C01826=1232.240,4.980,-41.243,-179.381,5.306,148.733
C01827=1232.235,5.230,-41.257,-179.378,5.306,148.732
C01828=1232.230,5.479,-41.273,-179.376,5.307,148.732
C01829=1232.225,5.729,-41.287,-179.373,5.306,148.731
C01830=1232.220,5.979,-41.301,-179.371,5.307,148.730
C01831=1232.215,6.228,-41.316,-179.368,5.308,148.730
C01832=1232.210,6.478,-41.331,-179.366,5.307,148.729
C01833=1232.205,6.727,-41.346,-179.363,5.308,148.728
C01834=1232.200,6.977,-41.361,-179.361,5.308,148.728
C01835=1232.195,7.226,-41.376,-179.358,5.309,148.727
C01836=1232.190,7.476,-41.390,-179.356,5.309,148.726
C01837=1232.185,7.725,-41.405,-179.353,5.309,148.726
C01838=1232.180,7.975,-41.420,-179.351,5.310,148.725
C01839=1232.175,8.224,-41.435,-179.348,5.310,148.724
C01840=1232.170,8.474,-41.450,-179.345,5.310,148.723
C01841=1232.165,8.723,-41.465,-179.343,5.310,148.723
C01842=1232.159,8.973,-41.479,-179.340,5.311,148.722
C01843=1232.155,9.222,-41.494,-179.338,5.311,148.721
C01844=1232.150,9.472,-41.509,-179.335,5.311,148.721
C01845=1232.144,9.721,-41.524,-179.333,5.311,148.720
C01846=1232.140,9.970,-41.539,-179.330,5.312,148.719
C01847=1232.135,10.220,-41.554,-179.328,5.312,148.719
C01848=1232.129,10.469,-41.569,-179.325,5.312,148.718
C01849=1232.124,10.719,-41.583,-179.323,5.313,148.717
C01850=1232.120,10.968,-41.598,-179.320,5.313,148.716
C01851=1232.114,11.217,-41.614,-179.318,5.313,148.716
C01852=1232.109,11.467,-41.628,-179.315,5.314,148.715
C01853=1232.105,11.717,-41.644,-179.313,5.314,148.714
C01854=1232.100,11.967,-41.658,-179.310,5.315,148.714
C01855=1232.095,12.216,-41.673,-179.308,5.314,148.713
C01856=1232.090,12.465,-41.689,-179.305,5.315,148.712
C01857=1232.085,12.715,-41.703,-179.303,5.315,148.712
C01858=1232.079,12.965,-41.719,-179.300,5.316,148.711
C01859=1232.075,13.214,-41.734,-179.298,5.316,148.710
C01860=1232.070,13.463,-41.748,-179.295,5.316,148.710
C01861=1232.064,13.713,-41.764,-179.293,5.317,148.709
C01862=1232.060,13.962,-41.779,-179.290,5.317,148.708
C01863=1232.054,14.212,-41.794,-179.287,5.318,148.708
C01864=1232.050,14.462,-41.809,-179.285,5.318,148.707
C01865=1232.045,14.711,-41.825,-179.283,5.318,148.706
C01866=1232.040,14.960,-41.840,-179.280,5.319,148.705
C01867=1232.034,15.210,-41.854,-179.277,5.319,148.705
C01868=1232.030,15.459,-41.869,-179.275,5.319,148.704
C01869=1232.024,15.709,-41.885,-179.273,5.320,148.703
C01870=1232.020,15.958,-41.900,-179.270,5.320,148.703
C01871=1232.014,16.209,-41.915,-179.267,5.321,148.702
C01872=1232.010,16.458,-41.930,-179.265,5.320,148.701
C01873=1232.004,16.707,-41.946,-179.263,5.321,148.701
C01874=1232.000,16.956,-41.961,-179.260,5.321,148.700
C01875=1231.994,17.206,-41.976,-179.257,5.322,148.699
C01876=1231.989,17.455,-41.991,-179.255,5.322,148.699
C01877=1231.984,17.705,-42.006,-179.253,5.322,148.698
C01878=1231.980,17.954,-42.022,-179.250,5.323,148.697
C01879=1231.975,18.204,-42.037,-179.248,5.324,148.697
C01880=1231.970,18.453,-42.052,-179.245,5.324,148.696
C01881=1231.964,18.703,-42.067,-179.243,5.324,148.695
C01882=1231.960,18.952,-42.082,-179.240,5.324,148.695
C01883=1231.955,19.202,-42.098,-179.238,5.325,148.694
C01884=1231.950,19.451,-42.113,-179.235,5.326,148.693
C01885=1231.945,19.701,-42.129,-179.233,5.325,148.693
C01886=1231.940,19.950,-42.144,-179.230,5.326,148.692
C01887=1231.935,20.199,-42.159,-179.228,5.326,148.691
C01888=1231.930,20.449,-42.175,-179.225,5.327,148.691
C01889=1231.925,20.699,-42.189,-179.223,5.328,148.690
C01890=1231.920,20.948,-42.205,-179.220,5.327,148.689
C01891=1231.915,21.197,-42.220,-179.218,5.328,148.689
C01892=1231.910,21.447,-42.236,-179.215,5.328,148.688
C01893=1231.905,21.697,-42.252,-179.213,5.329,148.687
C01894=1231.900,21.946,-42.267,-179.210,5.329,148.687
C01895=1231.895,22.195,-42.282,-179.208,5.329,148.686
C01896=1231.890,22.445,-42.297,-179.205,5.330,148.685
C01897=1231.885,22.695,-42.313,-179.202,5.330,148.685
C01898=1231.880,22.944,-42.329,-179.200,5.331,148.684
C01899=1231.875,23.193,-42.344,-179.198,5.331,148.683
C01900=1231.870,23.443,-42.359,-179.195,5.331,148.683
C01901=1231.865,23.693,-42.375,-179.192,5.332,148.682
C01902=1231.861,23.942,-42.390,-179.190,5.332,148.681
C01903=1231.855,24.191,-42.406,-179.187,5.333,148.680
C01904=1231.850,24.441,-42.421,-179.185,5.332,148.680
C01905=1231.846,24.690,-42.437,-179.182,5.333,148.679
C01906=1231.840,24.940,-42.452,-179.180,5.334,148.678
C01907=1231.835,25.189,-42.468,-179.177,5.334,148.678
C01908=1231.830,25.438,-42.483,-179.175,5.335,148.677
C01909=1231.825,25.688,-42.499,-179.172,5.334,148.676
C01910=1231.820,25.938,-42.514,-179.170,5.335,148.676
C01911=1231.815,26.187,-42.529,-179.167,5.336,148.675
C01912=1231.811,26.437,-42.545,-179.165,5.336,148.674
C01913=1231.806,26.686,-42.562,-179.162,5.337,148.674
C01914=1231.800,26.935,-42.577,-179.160,5.336,148.673
C01915=1231.796,27.184,-42.592,-179.157,5.337,148.672
C01916=1231.791,27.434,-42.608,-179.155,5.337,148.672
C01917=1231.785,27.684,-42.624,-179.152,5.338,148.671
C01918=1231.780,27.933,-42.639,-179.149,5.339,148.670
C01919=1231.776,28.183,-42.655,-179.147,5.338,148.670
C01920=1231.771,28.432,-42.670,-179.145,5.339,148.669
C01921=1231.765,28.681,-42.687,-179.142,5.339,148.668
C01922=1231.761,28.931,-42.703,-179.140,5.340,148.668
C01923=1231.756,29.180,-42.718,-179.137,5.341,148.667
C01924=1231.750,29.449,-42.735,-179.134,5.341,148.666
C01925=1231.745,29.717,-42.752,-179.131,5.342,148.666
C01926=1231.740,29.986,-42.769,-179.129,5.342,148.665
C01927=1231.734,30.255,-42.786,-179.126,5.343,148.664
C01928=1231.729,30.504,-42.802,-179.124,5.342,148.663
C01929=1231.724,30.753,-42.817,-179.121,5.343,148.663
C01930=1231.720,31.003,-42.833,-179.119,5.344,148.662
C01931=1231.715,31.252,-42.849,-179.116,5.344,148.661
C01932=1231.710,31.502,-42.865,-179.113,5.345,148.661
C01933=1231.704,31.752,-42.880,-179.111,5.345,148.660
C01934=1231.699,32.001,-42.896,-179.109,5.345,148.659
C01935=1231.695,32.250,-42.912,-179.106,5.346,148.659
C01936=1231.690,32.500,-42.928,-179.103,5.346,148.658
C01937=1231.684,32.749,-42.943,-179.101,5.347,148.657
C01938=1231.680,32.999,-42.959,-179.098,5.347,148.657
C01939=1231.675,33.248,-42.976,-179.095,5.348,148.656
C01940=1231.670,33.498,-42.991,-179.093,5.348,148.655
C01941=1231.664,33.748,-43.007,-179.091,5.348,148.655
C01942=1231.660,33.996,-43.023,-179.089,5.349,148.654
C01943=1231.655,34.246,-43.039,-179.086,5.350,148.654
C01944=1231.650,34.496,-43.054,-179.083,5.350,148.653
C01945=1231.645,34.745,-43.071,-179.081,5.351,148.652
C01946=1231.640,34.994,-43.087,-179.079,5.350,148.652
C01947=1231.636,35.244,-43.103,-179.076,5.351,148.651
C01948=1231.630,35.493,-43.119,-179.073,5.352,148.650
C01949=1231.625,35.743,-43.134,-179.071,5.352,148.649
C01950=1231.620,35.992,-43.151,-179.068,5.353,148.649
C01951=1231.615,36.242,-43.167,-179.065,5.353,148.648
C01952=1231.610,36.491,-43.183,-179.063,5.353,148.647
C01953=1231.605,36.740,-43.199,-179.061,5.354,148.647
C01954=1231.600,36.991,-43.215,-179.058,5.354,148.646
C01955=1231.596,37.239,-43.231,-179.055,5.355,148.645
C01956=1231.591,37.488,-43.246,-179.053,5.355,148.645
C01957=1231.586,37.738,-43.263,-179.050,5.356,148.644
C01958=1231.581,37.987,-43.278,-179.047,5.356,148.643
C01959=1231.576,38.237,-43.295,-179.045,5.356,148.643
C01960=1231.571,38.486,-43.311,-179.043,5.357,148.642
C01961=1231.566,38.736,-43.327,-179.041,5.358,148.642
C01962=1231.561,38.985,-43.343,-179.038,5.358,148.641
C01963=1231.556,39.235,-43.360,-179.035,5.359,148.640
C01964=1231.551,39.484,-43.375,-179.033,5.359,148.640
C01965=1231.547,39.733,-43.392,-179.030,5.360,148.639
C01966=1231.541,39.983,-43.407,-179.028,5.360,148.638
C01967=1231.537,40.232,-43.424,-179.025,5.360,148.638
C01968=1231.531,40.482,-43.440,-179.023,5.361,148.637
C01969=1231.526,40.732,-43.457,-179.020,5.361,148.636
C01970=1231.521,40.981,-43.473,-179.017,5.362,148.636
C01971=1231.516,41.230,-43.489,-179.015,5.362,148.635
C01972=1231.511,41.480,-43.505,-179.012,5.363,148.634
C01973=1231.506,41.729,-43.522,-179.010,5.363,148.633
C01974=1231.501,41.978,-43.538,-179.008,5.364,148.633
C01975=1231.496,42.228,-43.554,-179.005,5.364,148.632
C01976=1231.491,42.477,-43.570,-179.003,5.365,148.632
C01977=1231.487,42.727,-43.586,-179.000,5.365,148.631
C01978=1231.482,42.976,-43.602,-178.997,5.366,148.630
C01979=1231.477,43.225,-43.619,-178.995,5.366,148.630
C01980=1231.472,43.475,-43.635,-178.992,5.367,148.629
C01981=1231.466,43.725,-43.652,-178.990,5.367,148.628
C01982=1231.462,43.974,-43.669,-178.987,5.367,148.628
C01983=1231.457,44.223,-43.684,-178.985,5.368,148.627
C01984=1231.452,44.473,-43.701,-178.982,5.368,148.626
C01985=1231.447,44.722,-43.717,-178.979,5.369,148.626
C01986=1231.442,44.972,-43.733,-178.977,5.370,148.625
C01987=1231.437,45.221,-43.749,-178.975,5.371,148.625
C01988=1231.433,45.470,-43.766,-178.972,5.371,148.624
C01989=1231.427,45.720,-43.782,-178.970,5.371,148.623
C01990=1231.422,45.969,-43.799,-178.967,5.371,148.623
C01991=1231.418,46.219,-43.816,-178.965,5.372,148.622
C01992=1231.413,46.468,-43.832,-178.962,5.373,148.621
C01993=1231.408,46.718,-43.848,-178.959,5.373,148.621
C01994=1231.403,46.966,-43.864,-178.957,5.374,148.620
C01995=1231.397,47.216,-43.881,-178.954,5.374,148.619
C01996=1231.393,47.466,-43.898,-178.951,5.375,148.618
C01997=1231.388,47.715,-43.914,-178.949,5.375,148.618
C01998=1231.383,47.965,-43.930,-178.947,5.376,148.617
C01999=1231.378,48.213,-43.947,-178.945,5.376,148.617
C02000=1231.373,48.463,-43.964,-178.942,5.377,148.616
C02001=1231.368,48.713,-43.981,-178.939,5.377,148.615
C02002=1231.363,48.961,-43.997,-178.937,5.378,148.615
C02003=1231.358,49.212,-44.013,-178.934,5.378,148.614
C02004=1231.353,49.461,-44.030,-178.931,5.379,148.613
C02005=1231.348,49.710,-44.046,-178.929,5.380,148.613
C02006=1231.344,49.960,-44.063,-178.926,5.380,148.612
C02007=1231.339,50.209,-44.080,-178.924,5.381,148.611
C02008=1231.333,50.458,-44.097,-178.921,5.382,148.611
C02009=1231.329,50.708,-44.113,-178.919,5.381,148.610
C02010=1231.323,50.957,-44.129,-178.917,5.382,148.610
C02011=1231.319,51.207,-44.145,-178.914,5.382,148.609
C02012=1231.314,51.456,-44.163,-178.911,5.383,148.608
C02013=1231.309,51.705,-44.179,-178.909,5.384,148.608
C02014=1231.304,51.955,-44.196,-178.906,5.384,148.607
C02015=1231.299,52.204,-44.213,-178.904,5.385,148.606
C02016=1231.295,52.454,-44.230,-178.901,5.385,148.606
C02017=1231.289,52.703,-44.246,-178.898,5.386,148.605
C02018=1231.285,52.952,-44.263,-178.896,5.387,148.604
C02019=1231.280,53.202,-44.280,-178.893,5.387,148.604
C02020=1231.275,53.451,-44.296,-178.891,5.387,148.603
C02021=1231.270,53.700,-44.313,-178.889,5.388,148.602
C02022=1231.265,53.950,-44.330,-178.886,5.388,148.602
C02023=1231.260,54.199,-44.346,-178.883,5.389,148.601
C02024=1231.255,54.448,-44.363,-178.881,5.389,148.600
C02025=1231.250,54.698,-44.380,-178.878,5.390,148.600
C02026=1231.246,54.948,-44.397,-178.876,5.391,148.599
C02027=1231.240,55.197,-44.414,-178.873,5.392,148.599
C02028=1231.235,55.465,-44.432,-178.871,5.392,148.598
C02029=1231.230,55.733,-44.450,-178.868,5.392,148.597
C02030=1231.224,56.003,-44.468,-178.865,5.393,148.596
C02031=1231.219,56.270,-44.485,-178.862,5.394,148.596
C02032=1231.214,56.520,-44.503,-178.860,5.394,148.595
C02033=1231.209,56.770,-44.519,-178.857,5.395,148.594
C02034=1231.204,57.019,-44.537,-178.855,5.396,148.594
C02035=1231.199,57.268,-44.554,-178.852,5.396,148.593
C02036=1231.195,57.517,-44.570,-178.850,5.397,148.593
C02037=1231.190,57.767,-44.588,-178.847,5.397,148.592
C02038=1231.185,58.016,-44.604,-178.844,5.398,148.591
C02039=1231.179,58.266,-44.621,-178.842,5.399,148.591
C02040=1231.175,58.515,-44.638,-178.839,5.399,148.590
C02041=1231.170,58.765,-44.655,-178.837,5.400,148.589
C02042=1231.165,59.014,-44.673,-178.834,5.401,148.589
C02043=1231.160,59.263,-44.689,-178.832,5.401,148.588
C02044=1231.155,59.512,-44.706,-178.830,5.401,148.588
C02045=1231.150,59.762,-44.723,-178.827,5.402,148.587
C02046=1231.145,60.012,-44.740,-178.824,5.402,148.586
C02047=1231.140,60.261,-44.757,-178.822,5.403,148.586
C02048=1231.136,60.510,-44.774,-178.819,5.403,148.585
C02049=1231.130,60.759,-44.792,-178.817,5.404,148.584
C02050=1231.126,61.009,-44.808,-178.814,5.405,148.584
C02051=1231.121,61.259,-44.826,-178.812,5.405,148.583
C02052=1231.116,61.507,-44.843,-178.809,5.406,148.582
C02053=1231.111,61.757,-44.860,-178.807,5.407,148.582
C02054=1231.106,62.006,-44.876,-178.804,5.407,148.581
C02055=1231.101,62.256,-44.894,-178.801,5.408,148.580
C02056=1231.097,62.505,-44.911,-178.799,5.409,148.580
C02057=1231.092,62.754,-44.928,-178.796,5.409,148.579
C02058=1231.087,63.004,-44.945,-178.794,5.410,148.579
C02059=1231.081,63.253,-44.962,-178.791,5.410,148.578
C02060=1231.077,63.502,-44.979,-178.789,5.411,148.577
C02061=1231.072,63.752,-44.997,-178.786,5.412,148.577
C02062=1231.067,64.002,-45.014,-178.783,5.412,148.576
C02063=1231.062,64.250,-45.031,-178.781,5.413,148.576
C02064=1231.057,64.500,-45.049,-178.779,5.414,148.575
C02065=1231.053,64.750,-45.065,-178.776,5.414,148.574
C02066=1231.047,64.998,-45.083,-178.773,5.415,148.574
C02067=1231.042,65.248,-45.100,-178.771,5.415,148.573
C02068=1231.038,65.497,-45.117,-178.768,5.416,148.572
C02069=1231.033,65.747,-45.135,-178.766,5.417,148.572
C02070=1231.028,65.996,-45.151,-178.763,5.418,148.571
C02071=1231.023,66.245,-45.169,-178.761,5.417,148.570
C02072=1231.018,66.495,-45.187,-178.759,5.418,148.570
C02073=1231.014,66.744,-45.204,-178.756,5.418,148.569
C02074=1231.009,66.994,-45.221,-178.753,5.419,148.569
C02075=1231.003,67.243,-45.238,-178.751,5.420,148.568
C02076=1230.999,67.492,-45.256,-178.749,5.421,148.567
C02077=1230.993,67.741,-45.273,-178.746,5.421,148.567
C02078=1230.988,67.991,-45.291,-178.743,5.422,148.566
C02079=1230.984,68.240,-45.307,-178.741,5.422,148.565
C02080=1230.979,68.489,-45.325,-178.738,5.423,148.565
C02081=1230.974,68.739,-45.343,-178.735,5.423,148.564
C02082=1230.970,68.988,-45.360,-178.733,5.424,148.564
C02083=1230.964,69.238,-45.377,-178.731,5.425,148.563
C02084=1230.960,69.487,-45.395,-178.728,5.426,148.562
C02085=1230.954,69.737,-45.413,-178.725,5.426,148.562
C02086=1230.950,69.986,-45.430,-178.723,5.427,148.561
C02087=1230.945,70.235,-45.447,-178.721,5.428,148.561
C02088=1230.940,70.485,-45.465,-178.718,5.428,148.560
C02089=1230.935,70.733,-45.482,-178.715,5.429,148.559
C02090=1230.930,70.983,-45.500,-178.713,5.430,148.559
C02091=1230.925,71.232,-45.517,-178.710,5.430,148.558
C02092=1230.920,71.481,-45.535,-178.707,5.431,148.557
C02093=1230.916,71.730,-45.552,-178.705,5.432,148.557
C02094=1230.911,71.980,-45.569,-178.703,5.432,148.556
C02095=1230.906,72.229,-45.587,-178.700,5.433,148.556
C02096=1230.900,72.479,-45.605,-178.697,5.433,148.555
C02097=1230.895,72.728,-45.623,-178.695,5.434,148.554
C02098=1230.891,72.977,-45.640,-178.693,5.435,148.554
C02099=1230.886,73.227,-45.657,-178.690,5.436,148.553
C02100=1230.881,73.476,-45.675,-178.687,5.436,148.552
C02101=1230.876,73.725,-45.693,-178.685,5.437,148.552
C02102=1230.871,73.975,-45.710,-178.682,5.437,148.551
C02103=1230.867,74.224,-45.728,-178.680,5.438,148.550
C02104=1230.862,74.473,-45.746,-178.677,5.439,148.550
C02105=1230.857,74.723,-45.763,-178.675,5.439,148.549
C02106=1230.852,74.972,-45.781,-178.672,5.440,148.549
C02107=1230.847,75.221,-45.799,-178.669,5.441,148.548
C02108=1230.842,75.471,-45.816,-178.666,5.442,148.547
C02109=1230.838,75.720,-45.834,-178.664,5.443,148.547
C02110=1230.833,75.969,-45.852,-178.662,5.444,148.546
C02111=1230.828,76.218,-45.870,-178.659,5.444,148.546
C02112=1230.823,76.469,-45.887,-178.656,5.445,148.545
C02113=1230.818,76.718,-45.905,-178.654,5.445,148.544
C02114=1230.813,76.967,-45.923,-178.652,5.446,148.544
C02115=1230.808,77.216,-45.941,-178.649,5.447,148.543
C02116=1230.803,77.465,-45.959,-178.646,5.447,148.543
C02117=1230.799,77.715,-45.976,-178.644,5.448,148.542
C02118=1230.794,77.964,-45.994,-178.641,5.449,148.541
C02119=1230.789,78.213,-46.012,-178.639,5.450,148.541
C02120=1230.784,78.463,-46.030,-178.636,5.450,148.540
C02121=1230.779,78.712,-46.048,-178.634,5.451,148.540
C02122=1230.774,78.961,-46.065,-178.631,5.451,148.539
C02123=1230.769,79.211,-46.083,-178.628,5.452,148.538
C02124=1230.764,79.460,-46.101,-178.626,5.453,148.538
C02125=1230.759,79.709,-46.119,-178.624,5.454,148.537
C02126=1230.755,79.959,-46.137,-178.621,5.454,148.537
C02127=1230.750,80.208,-46.155,-178.618,5.455,148.536
C02128=1230.745,80.457,-46.173,-178.616,5.456,148.535
C02129=1230.740,80.707,-46.191,-178.614,5.456,148.535
C02130=1230.735,80.956,-46.209,-178.611,5.457,148.534
C02131=1230.730,81.205,-46.227,-178.608,5.457,148.533
C02132=1230.725,81.474,-46.246,-178.605,5.459,148.533
C02133=1230.720,81.742,-46.265,-178.603,5.460,148.532
C02134=1230.715,82.010,-46.285,-178.600,5.460,148.531
C02135=1230.710,82.278,-46.304,-178.597,5.461,148.531
C02136=1230.705,82.528,-46.322,-178.595,5.461,148.530
C02137=1230.700,82.777,-46.340,-178.593,5.462,148.530
C02138=1230.695,83.026,-46.358,-178.590,5.463,148.529
C02139=1230.691,83.276,-46.376,-178.587,5.463,148.528
C02140=1230.686,83.525,-46.394,-178.584,5.465,148.528
C02141=1230.681,83.774,-46.412,-178.582,5.466,148.527
C02142=1230.675,84.024,-46.431,-178.579,5.466,148.527
C02143=1230.670,84.273,-46.449,-178.577,5.467,148.526
C02144=1230.666,84.522,-46.467,-178.574,5.468,148.525
C02145=1230.661,84.772,-46.485,-178.572,5.469,148.525
C02146=1230.656,85.021,-46.503,-178.569,5.469,148.524
C02147=1230.651,85.270,-46.521,-178.567,5.470,148.524
C02148=1230.646,85.519,-46.539,-178.564,5.470,148.523
C02149=1230.642,85.769,-46.557,-178.562,5.471,148.523
C02150=1230.637,86.018,-46.575,-178.559,5.472,148.522
C02151=1230.632,86.268,-46.594,-178.557,5.473,148.521
C02152=1230.627,86.517,-46.612,-178.554,5.473,148.521
C02153=1230.622,86.766,-46.630,-178.551,5.474,148.520
C02154=1230.617,87.015,-46.648,-178.549,5.476,148.520
C02155=1230.612,87.265,-46.666,-178.546,5.476,148.519
C02156=1230.608,87.514,-46.685,-178.544,5.477,148.518
C02157=1230.603,87.763,-46.703,-178.541,5.477,148.518
C02158=1230.598,88.012,-46.721,-178.539,5.478,148.517
C02159=1230.593,88.261,-46.739,-178.536,5.479,148.517
C02160=1230.588,88.512,-46.758,-178.534,5.480,148.516
C02161=1230.583,88.761,-46.776,-178.531,5.480,148.515
C02162=1230.579,89.009,-46.795,-178.529,5.481,148.515
C02163=1230.574,89.259,-46.813,-178.526,5.482,148.514
C02164=1230.569,89.508,-46.831,-178.524,5.482,148.513
C02165=1230.564,89.758,-46.849,-178.521,5.484,148.513
C02166=1230.559,90.007,-46.868,-178.518,5.485,148.512
C02167=1230.554,90.256,-46.886,-178.516,5.485,148.512
C02168=1230.550,90.505,-46.905,-178.513,5.486,148.511
C02169=1230.545,90.755,-46.923,-178.511,5.487,148.511
C02170=1230.539,91.004,-46.941,-178.508,5.487,148.510
C02171=1230.535,91.253,-46.960,-178.506,5.488,148.509
C02172=1230.530,91.503,-46.978,-178.503,5.489,148.509
C02173=1230.526,91.752,-46.996,-178.501,5.490,148.508
C02174=1230.520,92.001,-47.015,-178.498,5.490,148.508
C02175=1230.515,92.250,-47.033,-178.495,5.492,148.507
C02176=1230.511,92.500,-47.052,-178.492,5.492,148.506
C02177=1230.506,92.749,-47.070,-178.490,5.493,148.506
C02178=1230.501,92.998,-47.089,-178.488,5.494,148.505
C02179=1230.496,93.248,-47.107,-178.485,5.494,148.505
C02180=1230.491,93.497,-47.125,-178.483,5.495,148.504
C02181=1230.487,93.745,-47.144,-178.480,5.496,148.504
C02182=1230.482,93.996,-47.163,-178.478,5.497,148.503
C02183=1230.477,94.244,-47.182,-178.475,5.497,148.502
C02184=1230.472,94.493,-47.200,-178.472,5.499,148.502
C02185=1230.467,94.743,-47.219,-178.470,5.500,148.501
C02186=1230.463,94.992,-47.237,-178.467,5.500,148.501
C02187=1230.458,95.241,-47.255,-178.465,5.501,148.500
C02188=1230.453,95.491,-47.274,-178.462,5.502,148.500
C02189=1230.448,95.740,-47.293,-178.460,5.502,148.499
C02190=1230.443,95.989,-47.311,-178.457,5.503,148.498
C02191=1230.438,96.239,-47.331,-178.455,5.504,148.498
C02192=1230.434,96.488,-47.349,-178.452,5.505,148.497
C02193=1230.429,96.736,-47.367,-178.449,5.506,148.497
C02194=1230.424,96.987,-47.386,-178.447,5.507,148.496
C02195=1230.419,97.235,-47.405,-178.445,5.508,148.495
C02196=1230.414,97.485,-47.423,-178.442,5.508,148.495
C02197=1230.410,97.734,-47.443,-178.439,5.509,148.494
C02198=1230.405,97.983,-47.461,-178.437,5.510,148.494
C02199=1230.400,98.233,-47.480,-178.434,5.511,148.493
C02200=1230.395,98.482,-47.498,-178.431,5.512,148.492
C02201=1230.390,98.731,-47.517,-178.429,5.513,148.492
C02202=1230.385,98.981,-47.536,-178.427,5.513,148.491
C02203=1230.381,99.229,-47.555,-178.424,5.514,148.491
C02204=1230.375,99.479,-47.573,-178.421,5.515,148.490
C02205=1230.371,99.728,-47.592,-178.419,5.516,148.490
C02206=1230.365,99.977,-47.611,-178.416,5.517,148.489
C02207=1230.361,100.227,-47.630,-178.413,5.518,148.488
C02208=1230.356,100.475,-47.649,-178.411,5.519,148.488
C02209=1230.352,100.725,-47.667,-178.409,5.519,148.487
C02210=1230.346,100.974,-47.687,-178.406,5.520,148.487
C02211=1230.342,101.223,-47.705,-178.404,5.521,148.486
C02212=1230.337,101.473,-47.724,-178.401,5.521,148.486
C02213=1230.332,101.721,-47.743,-178.398,5.523,148.485
C02214=1230.327,101.972,-47.762,-178.396,5.524,148.485
C02215=1230.323,102.220,-47.781,-178.393,5.524,148.484
C02216=1230.318,102.470,-47.800,-178.391,5.525,148.483
C02217=1230.313,102.719,-47.818,-178.389,5.526,148.483
C02218=1230.308,102.968,-47.838,-178.386,5.527,148.482
C02219=1230.304,103.217,-47.857,-178.383,5.528,148.482
C02220=1230.298,103.467,-47.875,-178.380,5.529,148.481
C02221=1230.294,103.716,-47.894,-178.378,5.530,148.480
C02222=1230.289,103.965,-47.914,-178.376,5.530,148.480
C02223=1230.285,104.214,-47.933,-178.373,5.531,148.479
C02224=1230.279,104.463,-47.951,-178.371,5.532,148.479
C02225=1230.275,104.713,-47.970,-178.368,5.533,148.478
C02226=1230.270,104.962,-47.990,-178.365,5.534,148.478
C02227=1230.265,105.211,-48.009,-178.363,5.535,148.477
C02228=1230.260,105.460,-48.027,-178.360,5.535,148.476
C02229=1230.255,105.710,-48.047,-178.358,5.536,148.476
C02230=1230.251,105.958,-48.066,-178.356,5.537,148.475
C02231=1230.246,106.208,-48.085,-178.352,5.538,148.475
C02232=1230.240,106.458,-48.104,-178.350,5.539,148.474
C02233=1230.236,106.707,-48.123,-178.348,5.540,148.474
C02234=1230.231,106.956,-48.142,-178.345,5.541,148.473
C02235=1230.227,107.205,-48.161,-178.342,5.541,148.472
C02236=1230.221,107.473,-48.182,-178.340,5.543,148.472
C02237=1230.216,107.742,-48.202,-178.337,5.544,148.471
C02238=1230.211,108.010,-48.223,-178.334,5.544,148.471
C02239=1230.206,108.279,-48.244,-178.331,5.546,148.470
C02240=1230.202,108.528,-48.263,-178.329,5.546,148.469
C02241=1230.196,108.777,-48.282,-178.327,5.547,148.469
C02242=1230.192,109.026,-48.302,-178.324,5.548,148.468
C02243=1230.186,109.276,-48.321,-178.321,5.549,148.468
C02244=1230.182,109.525,-48.340,-178.319,5.550,148.467
C02245=1230.177,109.774,-48.359,-178.316,5.551,148.467
C02246=1230.172,110.024,-48.379,-178.313,5.552,148.466
C02247=1230.167,110.272,-48.397,-178.311,5.553,148.466
C02248=1230.162,110.522,-48.417,-178.308,5.554,148.465
C02249=1230.158,110.771,-48.437,-178.306,5.555,148.465
C02250=1230.153,111.020,-48.455,-178.303,5.556,148.464
C02251=1230.148,111.269,-48.475,-178.301,5.556,148.463
C02252=1230.143,111.518,-48.494,-178.299,5.557,148.463
C02253=1230.138,111.768,-48.514,-178.295,5.559,148.462
C02254=1230.134,112.017,-48.533,-178.293,5.559,148.462
C02255=1230.129,112.266,-48.552,-178.291,5.560,148.461
C02256=1230.124,112.516,-48.572,-178.288,5.561,148.461
C02257=1230.119,112.764,-48.591,-178.285,5.562,148.460
C02258=1230.115,113.014,-48.610,-178.283,5.563,148.460
C02259=1230.110,113.263,-48.630,-178.280,5.564,148.459
C02260=1230.105,113.512,-48.649,-178.278,5.565,148.458
C02261=1230.100,113.762,-48.669,-178.276,5.566,148.458
C02262=1230.095,114.011,-48.689,-178.272,5.567,148.457
C02263=1230.091,114.259,-48.708,-178.270,5.568,148.457
C02264=1230.086,114.509,-48.728,-178.268,5.569,148.456
C02265=1230.081,114.758,-48.747,-178.265,5.569,148.456
C02266=1230.076,115.007,-48.767,-178.262,5.571,148.455
C02267=1230.071,115.257,-48.786,-178.260,5.572,148.454
C02268=1230.067,115.505,-48.805,-178.258,5.573,148.454
C02269=1230.062,115.755,-48.825,-178.255,5.573,148.453
C02270=1230.057,116.004,-48.844,-178.252,5.574,148.453
C02271=1230.052,116.253,-48.864,-178.250,5.576,148.452
C02272=1230.048,116.502,-48.884,-178.247,5.576,148.452
C02273=1230.043,116.752,-48.904,-178.245,5.577,148.451
C02274=1230.037,117.001,-48.923,-178.242,5.578,148.451
C02275=1230.033,117.250,-48.942,-178.239,5.579,148.450
C02276=1230.029,117.499,-48.962,-178.237,5.580,148.450
C02277=1230.024,117.748,-48.982,-178.234,5.581,148.449
C02278=1230.019,117.997,-49.001,-178.232,5.582,148.448
C02279=1230.014,118.247,-49.021,-178.229,5.583,148.448
C02280=1230.009,118.496,-49.041,-178.227,5.584,148.447
C02281=1230.004,118.745,-49.061,-178.224,5.585,148.447
C02282=1230.000,118.994,-49.080,-178.222,5.586,148.446
C02283=1229.995,119.244,-49.100,-178.219,5.587,148.446
C02284=1229.990,119.493,-49.119,-178.217,5.588,148.445
C02285=1229.985,119.742,-49.140,-178.214,5.589,148.445
C02286=1229.980,119.991,-49.159,-178.212,5.590,148.444
C02287=1229.976,120.241,-49.179,-178.209,5.591,148.444
C02288=1229.971,120.489,-49.198,-178.207,5.592,148.443
C02289=1229.967,120.738,-49.218,-178.204,5.593,148.443
C02290=1229.962,120.988,-49.238,-178.201,5.593,148.442
C02291=1229.957,121.237,-49.258,-178.199,5.595,148.442
C02292=1229.952,121.486,-49.277,-178.196,5.596,148.441
C02293=1229.947,121.735,-49.297,-178.194,5.597,148.440
C02294=1229.943,121.984,-49.317,-178.191,5.598,148.440
C02295=1229.938,122.234,-49.337,-178.188,5.599,148.439
C02296=1229.933,122.482,-49.357,-178.186,5.600,148.439
C02297=1229.928,122.732,-49.377,-178.183,5.600,148.438
C02298=1229.924,122.981,-49.396,-178.181,5.602,148.438
C02299=1229.919,123.230,-49.417,-178.178,5.603,148.437
C02300=1229.914,123.479,-49.436,-178.176,5.604,148.437
C02301=1229.909,123.728,-49.457,-178.173,5.604,148.436
C02302=1229.904,123.978,-49.477,-178.170,5.606,148.435
C02303=1229.899,124.227,-49.497,-178.168,5.607,148.435
C02304=1229.895,124.476,-49.517,-178.166,5.608,148.434
C02305=1229.890,124.725,-49.537,-178.163,5.609,148.434
C02306=1229.885,124.974,-49.556,-178.160,5.610,148.433
C02307=1229.880,125.224,-49.576,-178.158,5.611,148.433
C02308=1229.876,125.473,-49.596,-178.156,5.612,148.432
C02309=1229.871,125.722,-49.617,-178.152,5.613,148.432
C02310=1229.866,125.970,-49.636,-178.150,5.614,148.431
C02311=1229.862,126.219,-49.656,-178.148,5.615,148.431
C02312=1229.857,126.469,-49.676,-178.145,5.616,148.430
C02313=1229.852,126.718,-49.696,-178.142,5.617,148.430
C02314=1229.847,126.968,-49.717,-178.140,5.618,148.429
C02315=1229.842,127.217,-49.737,-178.138,5.619,148.429
C02316=1229.838,127.466,-49.757,-178.135,5.620,148.428
C02317=1229.833,127.715,-49.777,-178.132,5.621,148.428
C02318=1229.828,127.964,-49.797,-178.130,5.622,148.427
C02319=1229.823,128.213,-49.817,-178.127,5.624,148.427
C02320=1229.819,128.462,-49.837,-178.124,5.624,148.426
C02321=1229.814,128.712,-49.857,-178.122,5.625,148.426
C02322=1229.809,128.961,-49.878,-178.119,5.627,148.425
C02323=1229.805,129.210,-49.898,-178.117,5.628,148.425
C02324=1229.799,129.459,-49.917,-178.114,5.628,148.424
C02325=1229.795,129.708,-49.938,-178.112,5.630,148.424
C02326=1229.790,129.957,-49.959,-178.109,5.631,148.423
C02327=1229.785,130.206,-49.978,-178.107,5.631,148.422
C02328=1229.781,130.455,-49.999,-178.104,5.632,148.422
C02329=1229.776,130.704,-50.019,-178.101,5.634,148.421
C02330=1229.771,130.954,-50.039,-178.099,5.635,148.421
C02331=1229.766,131.203,-50.060,-178.097,5.635,148.420
C02332=1229.762,131.452,-50.080,-178.094,5.637,148.420
C02333=1229.757,131.701,-50.100,-178.091,5.638,148.419
C02334=1229.752,131.950,-50.120,-178.089,5.639,148.419
C02335=1229.747,132.199,-50.141,-178.086,5.640,148.418
C02336=1229.742,132.448,-50.161,-178.084,5.641,148.418
C02337=1229.738,132.697,-50.181,-178.081,5.642,148.417
C02338=1229.733,132.947,-50.201,-178.079,5.644,148.417
C02339=1229.728,133.196,-50.222,-178.076,5.644,148.416
C02340=1229.723,133.464,-50.244,-178.073,5.646,148.416
C02341=1229.718,133.734,-50.266,-178.071,5.647,148.415
C02342=1229.713,134.002,-50.288,-178.068,5.648,148.415
C02343=1229.707,134.271,-50.310,-178.065,5.649,148.414
C02344=1229.703,134.520,-50.330,-178.063,5.650,148.413
C02345=1229.698,134.769,-50.351,-178.060,5.651,148.413
C02346=1229.693,135.018,-50.372,-178.058,5.652,148.412
C02347=1229.689,135.267,-50.392,-178.055,5.653,148.412
C02348=1229.684,135.516,-50.412,-178.052,5.655,148.411
C02349=1229.679,135.765,-50.433,-178.050,5.655,148.411
C02350=1229.675,136.014,-50.454,-178.047,5.657,148.410
C02351=1229.670,136.264,-50.473,-178.044,5.658,148.410
C02352=1229.665,136.513,-50.494,-178.042,5.659,148.409
C02353=1229.660,136.762,-50.515,-178.039,5.660,148.409
C02354=1229.656,137.011,-50.535,-178.037,5.661,148.408
C02355=1229.651,137.260,-50.556,-178.034,5.662,148.408
C02356=1229.646,137.509,-50.576,-178.032,5.664,148.407
C02357=1229.641,137.758,-50.597,-178.029,5.664,148.407
C02358=1229.637,138.007,-50.618,-178.027,5.665,148.406
C02359=1229.632,138.256,-50.638,-178.024,5.667,148.406
C02360=1229.627,138.506,-50.659,-178.022,5.668,148.405
C02361=1229.623,138.754,-50.680,-178.019,5.669,148.405
C02362=1229.618,139.004,-50.700,-178.017,5.670,148.404
C02363=1229.613,139.253,-50.721,-178.014,5.671,148.404
C02364=1229.608,139.502,-50.742,-178.011,5.673,148.403
C02365=1229.604,139.751,-50.762,-178.009,5.673,148.403
C02366=1229.599,140.000,-50.783,-178.007,5.674,148.402
C02367=1229.594,140.249,-50.804,-178.003,5.676,148.402
C02368=1229.589,140.498,-50.824,-178.001,5.677,148.401
C02369=1229.584,140.747,-50.845,-177.999,5.678,148.401
C02370=1229.580,140.996,-50.865,-177.996,5.679,148.400
C02371=1229.576,141.246,-50.887,-177.993,5.680,148.400
C02372=1229.571,141.495,-50.908,-177.991,5.682,148.399
C02373=1229.566,141.744,-50.929,-177.988,5.682,148.399
C02374=1229.562,141.993,-50.949,-177.986,5.683,148.398
C02375=1229.556,142.242,-50.970,-177.983,5.685,148.398
C02376=1229.552,142.491,-50.990,-177.981,5.686,148.397
C02377=1229.547,142.740,-51.011,-177.978,5.688,148.397
C02378=1229.543,142.989,-51.032,-177.976,5.688,148.396
C02379=1229.537,143.238,-51.053,-177.973,5.689,148.396
C02380=1229.532,143.487,-51.074,-177.970,5.691,148.395
C02381=1229.528,143.736,-51.095,-177.968,5.692,148.395
C02382=1229.523,143.986,-51.116,-177.966,5.692,148.394
C02383=1229.519,144.235,-51.136,-177.963,5.694,148.394
C02384=1229.514,144.484,-51.158,-177.960,5.695,148.393
C02385=1229.510,144.733,-51.178,-177.958,5.697,148.393
C02386=1229.504,144.982,-51.199,-177.955,5.697,148.392
C02387=1229.499,145.231,-51.220,-177.953,5.698,148.392
C02388=1229.495,145.479,-51.241,-177.950,5.700,148.391
C02389=1229.490,145.729,-51.263,-177.948,5.701,148.391
C02390=1229.486,145.978,-51.283,-177.945,5.703,148.390
C02391=1229.481,146.227,-51.305,-177.942,5.703,148.390
C02392=1229.476,146.476,-51.326,-177.940,5.705,148.389
C02393=1229.472,146.725,-51.346,-177.937,5.706,148.389
C02394=1229.466,146.974,-51.367,-177.935,5.707,148.388
C02395=1229.462,147.224,-51.389,-177.932,5.708,148.388
C02396=1229.458,147.473,-51.410,-177.930,5.709,148.387
C02397=1229.453,147.722,-51.431,-177.927,5.711,148.387
C02398=1229.448,147.971,-51.452,-177.925,5.712,148.386
C02399=1229.443,148.220,-51.473,-177.922,5.713,148.386
C02400=1229.438,148.468,-51.494,-177.919,5.714,148.385
C02401=1229.434,148.718,-51.516,-177.917,5.715,148.385
C02402=1229.429,148.967,-51.536,-177.914,5.717,148.384
C02403=1229.424,149.216,-51.558,-177.912,5.718,148.384
C02404=1229.419,149.465,-51.579,-177.909,5.719,148.383
C02405=1229.415,149.713,-51.600,-177.907,5.720,148.383
C02406=1229.411,149.963,-51.621,-177.904,5.721,148.382
C02407=1229.405,150.213,-51.642,-177.901,5.723,148.382
C02408=1229.401,150.461,-51.664,-177.899,5.724,148.382
C02409=1229.396,150.710,-51.684,-177.896,5.725,148.381
C02410=1229.392,150.959,-51.706,-177.894,5.726,148.381
C02411=1229.387,151.209,-51.727,-177.891,5.728,148.380
C02412=1229.382,151.457,-51.749,-177.889,5.729,148.380
C02413=1229.377,151.706,-51.769,-177.887,5.730,148.379
C02414=1229.373,151.956,-51.791,-177.884,5.731,148.379
C02415=1229.368,152.205,-51.812,-177.881,5.732,148.378
C02416=1229.363,152.454,-51.834,-177.878,5.734,148.378
C02417=1229.359,152.703,-51.854,-177.876,5.735,148.377
C02418=1229.354,152.952,-51.876,-177.873,5.736,148.377
C02419=1229.349,153.201,-51.897,-177.871,5.737,148.376
C02420=1229.344,153.450,-51.919,-177.868,5.739,148.376
C02421=1229.339,153.698,-51.941,-177.866,5.739,148.375
C02422=1229.335,153.948,-51.962,-177.863,5.741,148.375
C02423=1229.331,154.197,-51.983,-177.860,5.742,148.374
C02424=1229.326,154.446,-52.004,-177.858,5.743,148.374
C02425=1229.321,154.695,-52.026,-177.856,5.745,148.373
C02426=1229.316,154.944,-52.048,-177.853,5.745,148.373
C02427=1229.311,155.193,-52.069,-177.850,5.747,148.372
C02428=1229.306,155.442,-52.090,-177.848,5.748,148.372
C02429=1229.302,155.691,-52.112,-177.845,5.750,148.371
C02430=1229.298,155.940,-52.133,-177.843,5.751,148.371
C02431=1229.293,156.189,-52.154,-177.840,5.752,148.371
C02432=1229.289,156.438,-52.177,-177.838,5.753,148.370
C02433=1229.283,156.687,-52.198,-177.835,5.755,148.370
C02434=1229.278,156.936,-52.219,-177.833,5.756,148.369
C02435=1229.274,157.185,-52.241,-177.830,5.758,148.369
C02436=1229.269,157.435,-52.262,-177.827,5.758,148.368
C02437=1229.264,157.683,-52.284,-177.825,5.760,148.368
C02438=1229.260,157.933,-52.306,-177.823,5.761,148.367
C02439=1229.255,158.181,-52.328,-177.819,5.762,148.367
C02440=1229.250,158.430,-52.349,-177.817,5.763,148.366
C02441=1229.246,158.679,-52.370,-177.814,5.765,148.366
C02442=1229.241,158.928,-52.392,-177.812,5.766,148.365
C02443=1229.237,159.177,-52.413,-177.810,5.767,148.365
C02444=1229.232,159.447,-52.437,-177.807,5.768,148.364
C02445=1229.226,159.716,-52.460,-177.804,5.770,148.364
C02446=1229.222,159.985,-52.484,-177.801,5.772,148.363
C02447=1229.216,160.254,-52.507,-177.798,5.772,148.363
C02448=1229.211,160.503,-52.529,-177.796,5.774,148.362
C02449=1229.207,160.752,-52.551,-177.794,5.775,148.362
C02450=1229.202,161.001,-52.573,-177.790,5.777,148.361
C02451=1229.197,161.249,-52.594,-177.788,5.778,148.361
C02452=1229.193,161.499,-52.616,-177.786,5.780,148.361
C02453=1229.188,161.748,-52.637,-177.783,5.780,148.360
C02454=1229.184,161.997,-52.659,-177.780,5.782,148.360
C02455=1229.179,162.246,-52.681,-177.778,5.783,148.359
C02456=1229.174,162.494,-52.703,-177.775,5.785,148.359
C02457=1229.170,162.744,-52.725,-177.773,5.786,148.358
C02458=1229.165,162.992,-52.747,-177.770,5.787,148.358
C02459=1229.161,163.242,-52.769,-177.768,5.788,148.357
C02460=1229.156,163.490,-52.790,-177.765,5.790,148.357
C02461=1229.151,163.740,-52.812,-177.763,5.791,148.356
C02462=1229.146,163.989,-52.835,-177.760,5.792,148.356
C02463=1229.142,164.238,-52.857,-177.758,5.793,148.356
C02464=1229.137,164.487,-52.878,-177.755,5.795,148.355
C02465=1229.132,164.735,-52.900,-177.753,5.796,148.355
C02466=1229.128,164.985,-52.922,-177.750,5.798,148.354
C02467=1229.123,165.233,-52.944,-177.747,5.798,148.354
C02468=1229.118,165.483,-52.966,-177.745,5.800,148.353
C02469=1229.114,165.731,-52.988,-177.742,5.802,148.353
C02470=1229.109,165.981,-53.010,-177.739,5.803,148.352
C02471=1229.104,166.230,-53.032,-177.737,5.805,148.352
C02472=1229.099,166.479,-53.054,-177.735,5.806,148.352
C02473=1229.095,166.728,-53.076,-177.732,5.807,148.351
C02474=1229.090,166.977,-53.098,-177.729,5.808,148.351
C02475=1229.085,167.226,-53.119,-177.727,5.810,148.350
C02476=1229.081,167.475,-53.143,-177.724,5.811,148.350
C02477=1229.076,167.723,-53.164,-177.722,5.812,148.349
C02478=1229.072,167.973,-53.186,-177.719,5.813,148.349
C02479=1229.067,168.221,-53.208,-177.716,5.815,148.348
C02480=1229.062,168.471,-53.230,-177.714,5.816,148.348
C02481=1229.057,168.720,-53.252,-177.712,5.818,148.348
C02482=1229.053,168.969,-53.274,-177.708,5.819,148.347
C02483=1229.049,169.218,-53.297,-177.706,5.820,148.347
C02484=1229.044,169.466,-53.319,-177.704,5.822,148.346
C02485=1229.039,169.716,-53.341,-177.701,5.823,148.346
C02486=1229.034,169.965,-53.363,-177.698,5.825,148.345
C02487=1229.030,170.214,-53.385,-177.696,5.826,148.345
C02488=1229.025,170.462,-53.408,-177.694,5.827,148.344
C02489=1229.020,170.712,-53.430,-177.691,5.828,148.344
C02490=1229.015,170.960,-53.452,-177.688,5.830,148.344
C02491=1229.011,171.210,-53.474,-177.686,5.832,148.343
C02492=1229.007,171.458,-53.497,-177.683,5.832,148.343
C02493=1229.001,171.707,-53.519,-177.681,5.834,148.342
C02494=1228.997,171.957,-53.541,-177.678,5.835,148.342
C02495=1228.992,172.205,-53.564,-177.675,5.837,148.341
C02496=1228.987,172.454,-53.586,-177.673,5.838,148.341
C02497=1228.983,172.703,-53.608,-177.671,5.840,148.340
C02498=1228.979,172.952,-53.631,-177.668,5.841,148.340
C02499=1228.974,173.201,-53.653,-177.665,5.842,148.340
C02500=1228.969,173.450,-53.675,-177.663,5.844,148.339
C02501=1228.965,173.699,-53.698,-177.661,5.845,148.339
C02502=1228.960,173.948,-53.720,-177.657,5.846,148.338
C02503=1228.955,174.197,-53.742,-177.655,5.847,148.338
C02504=1228.951,174.446,-53.765,-177.653,5.849,148.337
C02505=1228.945,174.695,-53.787,-177.650,5.851,148.337
C02506=1228.941,174.943,-53.810,-177.648,5.852,148.336
C02507=1228.936,175.193,-53.832,-177.645,5.854,148.336
C02508=1228.932,175.441,-53.855,-177.643,5.855,148.336
C02509=1228.928,175.690,-53.877,-177.640,5.856,148.335
C02510=1228.923,175.940,-53.900,-177.637,5.858,148.335
C02511=1228.918,176.188,-53.922,-177.635,5.859,148.334
C02512=1228.913,176.438,-53.945,-177.632,5.861,148.334
C02513=1228.909,176.686,-53.967,-177.630,5.861,148.333
C02514=1228.903,176.935,-53.990,-177.627,5.863,148.333
C02515=1228.899,177.184,-54.012,-177.624,5.865,148.333
C02516=1228.894,177.434,-54.035,-177.622,5.866,148.332
C02517=1228.890,177.682,-54.057,-177.619,5.868,148.332
C02518=1228.886,177.931,-54.079,-177.617,5.869,148.331
C02519=1228.881,178.180,-54.103,-177.614,5.870,148.331
C02520=1228.876,178.428,-54.125,-177.611,5.872,148.330
C02521=1228.871,178.678,-54.148,-177.609,5.873,148.330
C02522=1228.867,178.926,-54.171,-177.607,5.875,148.330
C02523=1228.862,179.175,-54.193,-177.604,5.876,148.329
C02524=1228.858,179.424,-54.216,-177.601,5.877,148.329
C02525=1228.853,179.674,-54.238,-177.599,5.879,148.328
C02526=1228.849,179.922,-54.261,-177.597,5.880,148.328
C02527=1228.844,180.171,-54.284,-177.594,5.882,148.328
C02528=1228.839,180.420,-54.306,-177.591,5.883,148.327
C02529=1228.835,180.669,-54.330,-177.589,5.885,148.327
C02530=1228.830,180.918,-54.353,-177.586,5.886,148.326
C02531=1228.825,181.167,-54.375,-177.584,5.887,148.326
C02532=1228.820,181.416,-54.398,-177.581,5.889,148.325
C02533=1228.816,181.665,-54.421,-177.578,5.891,148.325
C02534=1228.811,181.914,-54.443,-177.576,5.892,148.325
C02535=1228.807,182.162,-54.466,-177.573,5.894,148.324
C02536=1228.802,182.411,-54.489,-177.571,5.895,148.324
C02537=1228.797,182.660,-54.512,-177.568,5.896,148.323
C02538=1228.793,182.910,-54.534,-177.566,5.898,148.323
C02539=1228.788,183.158,-54.557,-177.563,5.899,148.323
C02540=1228.784,183.407,-54.580,-177.561,5.901,148.322
C02541=1228.779,183.656,-54.604,-177.558,5.902,148.322
C02542=1228.774,183.905,-54.626,-177.556,5.903,148.321
C02543=1228.770,184.154,-54.649,-177.553,5.905,148.321
C02544=1228.765,184.402,-54.672,-177.550,5.907,148.321
C02545=1228.760,184.652,-54.695,-177.548,5.908,148.320
C02546=1228.756,184.900,-54.718,-177.545,5.910,148.320
C02547=1228.751,185.150,-54.741,-177.542,5.911,148.319
C02548=1228.746,185.420,-54.766,-177.540,5.912,148.319
C02549=1228.742,185.688,-54.791,-177.537,5.914,148.318
C02550=1228.736,185.958,-54.816,-177.535,5.916,148.318
C02551=1228.731,186.228,-54.841,-177.531,5.917,148.317
C02552=1228.727,186.477,-54.864,-177.529,5.919,148.317
C02553=1228.722,186.726,-54.887,-177.527,5.920,148.317
C02554=1228.717,186.975,-54.910,-177.524,5.922,148.316
C02555=1228.713,187.223,-54.932,-177.521,5.924,148.316
C02556=1228.708,187.472,-54.956,-177.519,5.925,148.315
C02557=1228.703,187.722,-54.979,-177.516,5.926,148.315
C02558=1228.699,187.971,-55.002,-177.514,5.928,148.315
C02559=1228.695,188.219,-55.025,-177.511,5.929,148.314
C02560=1228.690,188.468,-55.048,-177.509,5.931,148.314
C02561=1228.685,188.717,-55.072,-177.506,5.933,148.313
C02562=1228.680,188.966,-55.095,-177.504,5.934,148.313
C02563=1228.676,189.214,-55.118,-177.501,5.935,148.313
C02564=1228.671,189.463,-55.141,-177.498,5.937,148.312
C02565=1228.667,189.712,-55.164,-177.496,5.939,148.312
C02566=1228.662,189.961,-55.188,-177.493,5.940,148.311
C02567=1228.657,190.211,-55.211,-177.490,5.942,148.311
C02568=1228.653,190.459,-55.234,-177.488,5.944,148.311
C02569=1228.649,190.708,-55.257,-177.486,5.945,148.310
C02570=1228.644,190.957,-55.280,-177.483,5.946,148.310
C02571=1228.639,191.206,-55.303,-177.480,5.948,148.309
C02572=1228.634,191.455,-55.327,-177.478,5.949,148.309
C02573=1228.629,191.703,-55.351,-177.475,5.951,148.309
C02574=1228.625,191.952,-55.374,-177.473,5.953,148.308
C02575=1228.621,192.201,-55.397,-177.470,5.954,148.308
C02576=1228.616,192.450,-55.420,-177.468,5.955,148.308
C02577=1228.611,192.699,-55.444,-177.465,5.957,148.307
C02578=1228.607,192.948,-55.467,-177.462,5.959,148.307
C02579=1228.602,193.197,-55.490,-177.460,5.960,148.306
C02580=1228.598,193.445,-55.514,-177.457,5.962,148.306
C02581=1228.593,193.694,-55.538,-177.455,5.964,148.306
C02582=1228.588,193.943,-55.561,-177.453,5.965,148.305
C02583=1228.583,194.192,-55.585,-177.449,5.966,148.305
C02584=1228.580,194.441,-55.607,-177.447,5.968,148.304
C02585=1228.575,194.690,-55.631,-177.445,5.969,148.304
C02586=1228.570,194.939,-55.655,-177.442,5.971,148.304
C02587=1228.566,195.188,-55.678,-177.439,5.973,148.303
C02588=1228.561,195.437,-55.701,-177.437,5.974,148.303
C02589=1228.557,195.685,-55.726,-177.434,5.975,148.302
C02590=1228.552,195.934,-55.749,-177.432,5.977,148.302
C02591=1228.547,196.183,-55.772,-177.429,5.979,148.302
C02592=1228.543,196.432,-55.796,-177.426,5.981,148.301
C02593=1228.538,196.681,-55.820,-177.424,5.982,148.301
C02594=1228.533,196.930,-55.843,-177.422,5.984,148.301
C02595=1228.529,197.179,-55.866,-177.419,5.985,148.300
C02596=1228.524,197.427,-55.890,-177.416,5.986,148.300
C02597=1228.520,197.676,-55.914,-177.414,5.988,148.299
C02598=1228.515,197.925,-55.937,-177.411,5.990,148.299
C02599=1228.511,198.174,-55.961,-177.409,5.992,148.299
C02600=1228.506,198.423,-55.985,-177.406,5.993,148.298
C02601=1228.501,198.672,-56.008,-177.404,5.995,148.298
C02602=1228.497,198.920,-56.032,-177.401,5.996,148.297
C02603=1228.492,199.169,-56.055,-177.398,5.998,148.297
C02604=1228.488,199.417,-56.080,-177.396,5.999,148.297
C02605=1228.483,199.667,-56.103,-177.393,6.001,148.296
C02606=1228.478,199.915,-56.128,-177.391,6.003,148.296
C02607=1228.473,200.164,-56.151,-177.388,6.005,148.296
C02608=1228.469,200.413,-56.175,-177.386,6.006,148.295
C02609=1228.464,200.662,-56.198,-177.383,6.007,148.295
C02610=1228.459,200.911,-56.222,-177.381,6.009,148.294
C02611=1228.455,201.159,-56.246,-177.378,6.011,148.294
C02612=1228.451,201.409,-56.269,-177.375,6.012,148.294
C02613=1228.446,201.657,-56.294,-177.373,6.014,148.293
C02614=1228.442,201.906,-56.317,-177.370,6.015,148.293
C02615=1228.437,202.155,-56.342,-177.368,6.017,148.293
C02616=1228.432,202.403,-56.366,-177.365,6.018,148.292
C02617=1228.428,202.653,-56.389,-177.363,6.020,148.292
C02618=1228.423,202.901,-56.413,-177.360,6.022,148.291
C02619=1228.418,203.150,-56.436,-177.358,6.024,148.291
C02620=1228.414,203.398,-56.461,-177.354,6.025,148.291
C02621=1228.409,203.648,-56.485,-177.352,6.026,148.290
C02622=1228.405,203.897,-56.509,-177.350,6.028,148.290
C02623=1228.400,204.145,-56.533,-177.347,6.030,148.290
C02624=1228.396,204.394,-56.556,-177.344,6.032,148.289
C02625=1228.391,204.643,-56.580,-177.342,6.033,148.289
C02626=1228.386,204.891,-56.605,-177.340,6.035,148.288
C02627=1228.381,205.140,-56.628,-177.337,6.037,148.288
C02628=1228.378,205.390,-56.653,-177.334,6.039,148.288
C02629=1228.373,205.638,-56.677,-177.332,6.040,148.287
C02630=1228.369,205.887,-56.700,-177.329,6.041,148.287
C02631=1228.363,206.136,-56.725,-177.327,6.043,148.287
C02632=1228.359,206.384,-56.749,-177.324,6.045,148.286
C02633=1228.355,206.634,-56.773,-177.321,6.047,148.286
C02634=1228.350,206.883,-56.797,-177.319,6.048,148.285
C02635=1228.345,207.131,-56.822,-177.317,6.050,148.285
C02636=1228.341,207.379,-56.846,-177.314,6.052,148.285
C02637=1228.336,207.628,-56.869,-177.311,6.053,148.284
C02638=1228.331,207.877,-56.894,-177.309,6.055,148.284
C02639=1228.327,208.126,-56.918,-177.307,6.056,148.284
C02640=1228.323,208.375,-56.942,-177.304,6.058,148.283
C02641=1228.318,208.623,-56.967,-177.301,6.060,148.283
C02642=1228.313,208.872,-56.990,-177.298,6.061,148.283
C02643=1228.309,209.122,-57.015,-177.296,6.063,148.282
C02644=1228.304,209.370,-57.039,-177.293,6.065,148.282
C02645=1228.300,209.619,-57.063,-177.291,6.066,148.281
C02646=1228.296,209.867,-57.087,-177.288,6.068,148.281
C02647=1228.290,210.116,-57.112,-177.286,6.070,148.281
C02648=1228.287,210.365,-57.137,-177.283,6.072,148.281
C02649=1228.281,210.614,-57.161,-177.280,6.074,148.280
C02650=1228.277,210.863,-57.185,-177.278,6.075,148.280
C02651=1228.272,211.111,-57.209,-177.276,6.077,148.279
C02652=1228.268,211.382,-57.236,-177.273,6.078,148.279
C02653=1228.263,211.652,-57.262,-177.270,6.080,148.279
C02654=1228.257,211.922,-57.289,-177.267,6.082,148.278
C02655=1228.252,212.193,-57.315,-177.264,6.085,148.278
C02656=1228.248,212.442,-57.340,-177.262,6.086,148.278
C02657=1228.244,212.691,-57.364,-177.259,6.087,148.277
C02658=1228.239,212.939,-57.388,-177.257,6.089,148.277
C02659=1228.235,213.188,-57.413,-177.254,6.091,148.277
C02660=1228.230,213.437,-57.437,-177.252,6.093,148.276
C02661=1228.225,213.686,-57.462,-177.249,6.095,148.276
C02662=1228.220,213.934,-57.486,-177.247,6.096,148.276
C02663=1228.216,214.183,-57.511,-177.244,6.098,148.275
C02664=1228.211,214.432,-57.535,-177.241,6.099,148.275
C02665=1228.207,214.681,-57.559,-177.238,6.101,148.274
C02666=1228.203,214.929,-57.585,-177.236,6.103,148.274
C02667=1228.198,215.178,-57.609,-177.233,6.105,148.274
C02668=1228.193,215.427,-57.634,-177.231,6.106,148.273
C02669=1228.189,215.676,-57.658,-177.229,6.108,148.273
C02670=1228.184,215.924,-57.683,-177.226,6.110,148.273
C02671=1228.180,216.173,-57.707,-177.223,6.111,148.272
C02672=1228.175,216.422,-57.732,-177.221,6.113,148.272
C02673=1228.171,216.671,-57.756,-177.218,6.115,148.272
C02674=1228.167,216.919,-57.782,-177.215,6.117,148.271
C02675=1228.162,217.168,-57.807,-177.213,6.118,148.271
C02676=1228.157,217.417,-57.831,-177.211,6.120,148.271
C02677=1228.153,217.666,-57.856,-177.208,6.122,148.270
C02678=1228.148,217.914,-57.880,-177.205,6.124,148.270
C02679=1228.143,218.162,-57.905,-177.203,6.126,148.270
C02680=1228.140,218.412,-57.930,-177.200,6.127,148.269
C02681=1228.135,218.660,-57.954,-177.198,6.129,148.269
C02682=1228.130,218.910,-57.979,-177.195,6.131,148.269
C02683=1228.126,219.158,-58.003,-177.193,6.132,148.268
C02684=1228.121,219.406,-58.029,-177.190,6.134,148.268
C02685=1228.116,219.656,-58.054,-177.188,6.136,148.268
C02686=1228.112,219.904,-58.078,-177.185,6.138,148.267
C02687=1228.108,220.153,-58.104,-177.182,6.140,148.267
C02688=1228.102,220.402,-58.128,-177.180,6.141,148.267
C02689=1228.099,220.651,-58.153,-177.177,6.143,148.266
C02690=1228.094,220.899,-58.178,-177.175,6.144,148.266
C02691=1228.089,221.148,-58.203,-177.172,6.146,148.266
C02692=1228.085,221.397,-58.227,-177.170,6.148,148.265
C02693=1228.080,221.645,-58.253,-177.167,6.150,148.265
C02694=1228.076,221.894,-58.278,-177.165,6.152,148.265
C02695=1228.071,222.143,-58.302,-177.162,6.154,148.264
C02696=1228.067,222.391,-58.327,-177.159,6.156,148.264
C02697=1228.062,222.640,-58.352,-177.157,6.157,148.264
C02698=1228.058,222.889,-58.377,-177.154,6.159,148.263
C02699=1228.053,223.137,-58.402,-177.152,6.160,148.263
C02700=1228.049,223.386,-58.428,-177.149,6.162,148.263
C02701=1228.044,223.635,-58.452,-177.147,6.164,148.262
C02702=1228.040,223.884,-58.477,-177.144,6.166,148.262
C02703=1228.035,224.132,-58.502,-177.141,6.168,148.262
C02704=1228.030,224.381,-58.527,-177.139,6.170,148.261
C02705=1228.026,224.630,-58.553,-177.136,6.172,148.261
C02706=1228.021,224.878,-58.577,-177.134,6.173,148.261
C02707=1228.017,225.127,-58.602,-177.132,6.175,148.261
C02708=1228.013,225.376,-58.627,-177.129,6.177,148.260
C02709=1228.008,225.624,-58.653,-177.127,6.178,148.260
C02710=1228.004,225.873,-58.679,-177.124,6.180,148.260
C02711=1227.999,226.122,-58.703,-177.121,6.182,148.259
C02712=1227.995,226.370,-58.728,-177.119,6.184,148.259
C02713=1227.990,226.619,-58.753,-177.116,6.186,148.259
C02714=1227.986,226.868,-58.779,-177.114,6.188,148.258
C02715=1227.981,227.117,-58.804,-177.111,6.190,148.258
C02716=1227.976,227.365,-58.829,-177.108,6.192,148.258
C02717=1227.972,227.614,-58.855,-177.106,6.193,148.257
C02718=1227.967,227.863,-58.880,-177.104,6.194,148.257
C02719=1227.962,228.111,-58.905,-177.101,6.196,148.257
C02720=1227.959,228.360,-58.930,-177.098,6.198,148.256
C02721=1227.954,228.609,-58.955,-177.096,6.200,148.256
C02722=1227.949,228.857,-58.981,-177.093,6.202,148.256
C02723=1227.945,229.106,-59.006,-177.091,6.204,148.255
C02724=1227.940,229.355,-59.031,-177.088,6.206,148.255
C02725=1227.936,229.603,-59.057,-177.086,6.208,148.255
C02726=1227.931,229.852,-59.082,-177.083,6.210,148.255
C02727=1227.927,230.100,-59.108,-177.081,6.212,148.254
C02728=1227.922,230.350,-59.133,-177.079,6.213,148.254
C02729=1227.917,230.598,-59.158,-177.076,6.215,148.254
C02730=1227.913,230.847,-59.184,-177.073,6.216,148.253
C02731=1227.909,231.096,-59.210,-177.071,6.218,148.253
C02732=1227.904,231.344,-59.235,-177.068,6.220,148.253
C02733=1227.900,231.593,-59.260,-177.065,6.222,148.252
C02734=1227.895,231.841,-59.286,-177.063,6.224,148.252
C02735=1227.890,232.090,-59.311,-177.061,6.226,148.252
C02736=1227.886,232.339,-59.337,-177.058,6.228,148.252
C02737=1227.881,232.587,-59.362,-177.055,6.230,148.251
C02738=1227.877,232.836,-59.388,-177.053,6.232,148.251
C02739=1227.873,233.085,-59.413,-177.050,6.234,148.251
C02740=1227.868,233.333,-59.439,-177.048,6.235,148.250
C02741=1227.864,233.582,-59.465,-177.045,6.236,148.250
C02742=1227.859,233.831,-59.490,-177.043,6.238,148.250
C02743=1227.855,234.079,-59.516,-177.040,6.240,148.249
C02744=1227.850,234.328,-59.541,-177.038,6.242,148.249
C02745=1227.846,234.577,-59.567,-177.035,6.244,148.249
C02746=1227.841,234.825,-59.592,-177.033,6.246,148.249
C02747=1227.837,235.074,-59.618,-177.030,6.248,148.248
C02748=1227.833,235.323,-59.643,-177.028,6.250,148.248
C02749=1227.828,235.571,-59.669,-177.025,6.252,148.248
C02750=1227.824,235.820,-59.694,-177.022,6.254,148.247
C02751=1227.819,236.069,-59.721,-177.020,6.256,148.247
C02752=1227.814,236.317,-59.746,-177.018,6.258,148.247
C02753=1227.809,236.566,-59.772,-177.015,6.260,148.247
C02754=1227.805,236.815,-59.798,-177.012,6.261,148.246
C02755=1227.801,237.063,-59.823,-177.010,6.263,148.246
C02756=1227.796,237.334,-59.852,-177.007,6.265,148.246
C02757=1227.791,237.606,-59.880,-177.005,6.267,148.245
C02758=1227.786,237.877,-59.908,-177.002,6.269,148.245
C02759=1227.782,238.148,-59.936,-176.999,6.272,148.245
C02760=1227.777,238.397,-59.962,-176.997,6.273,148.244
C02761=1227.772,238.646,-59.988,-176.994,6.275,148.244
C02762=1227.768,238.894,-60.014,-176.991,6.276,148.244
C02763=1227.763,239.143,-60.040,-176.989,6.278,148.243
C02764=1227.759,239.392,-60.065,-176.987,6.281,148.243
C02765=1227.754,239.640,-60.091,-176.984,6.282,148.243
C02766=1227.750,239.889,-60.118,-176.982,6.284,148.243
C02767=1227.746,240.137,-60.143,-176.979,6.286,148.242
C02768=1227.741,240.386,-60.169,-176.976,6.288,148.242
C02769=1227.736,240.634,-60.195,-176.974,6.290,148.242
C02770=1227.731,240.883,-60.221,-176.972,6.292,148.242
C02771=1227.728,241.132,-60.247,-176.969,6.294,148.241
C02772=1227.723,241.380,-60.273,-176.966,6.296,148.241
C02773=1227.719,241.629,-60.299,-176.964,6.298,148.241
C02774=1227.714,241.878,-60.325,-176.961,6.300,148.240
C02775=1227.710,242.126,-60.351,-176.959,6.302,148.240
C02776=1227.705,242.375,-60.377,-176.956,6.304,148.240
C02777=1227.700,242.624,-60.403,-176.954,6.306,148.240
C02778=1227.696,242.873,-60.429,-176.951,6.307,148.239
C02779=1227.692,243.121,-60.456,-176.948,6.309,148.239
C02780=1227.687,243.369,-60.482,-176.946,6.311,148.239
C02781=1227.683,243.618,-60.507,-176.944,6.313,148.239
C02782=1227.679,243.866,-60.534,-176.941,6.315,148.238
C02783=1227.674,244.115,-60.560,-176.938,6.317,148.238
C02784=1227.669,244.364,-60.586,-176.936,6.319,148.238
C02785=1227.666,244.612,-60.612,-176.933,6.321,148.237
C02786=1227.660,244.861,-60.638,-176.931,6.323,148.237
C02787=1227.656,245.109,-60.664,-176.929,6.325,148.237
C02788=1227.652,245.358,-60.691,-176.926,6.327,148.237
C02789=1227.647,245.607,-60.717,-176.923,6.329,148.236
C02790=1227.643,245.855,-60.743,-176.921,6.331,148.236
C02791=1227.638,246.104,-60.770,-176.919,6.333,148.236
C02792=1227.634,246.352,-60.796,-176.916,6.335,148.236
C02793=1227.630,246.601,-60.822,-176.913,6.337,148.235
C02794=1227.624,246.849,-60.848,-176.911,6.339,148.235
C02795=1227.620,247.098,-60.874,-176.909,6.341,148.235
C02796=1227.615,247.347,-60.901,-176.906,6.343,148.235
C02797=1227.611,247.595,-60.927,-176.903,6.344,148.234
C02798=1227.606,247.844,-60.954,-176.901,6.346,148.234
C02799=1227.603,248.092,-60.980,-176.898,6.348,148.234
C02800=1227.598,248.341,-61.006,-176.896,6.350,148.234
C02801=1227.594,248.590,-61.033,-176.893,6.352,148.233
C02802=1227.589,248.838,-61.060,-176.891,6.354,148.233
C02803=1227.585,249.087,-61.086,-176.888,6.356,148.233
C02804=1227.580,249.335,-61.113,-176.886,6.358,148.233
C02805=1227.576,249.584,-61.139,-176.883,6.360,148.232
C02806=1227.571,249.833,-61.166,-176.881,6.362,148.232
C02807=1227.567,250.080,-61.192,-176.878,6.364,148.232
C02808=1227.562,250.329,-61.218,-176.876,6.366,148.232
C02809=1227.558,250.577,-61.245,-176.873,6.368,148.231
C02810=1227.553,250.827,-61.271,-176.871,6.370,148.231
C02811=1227.549,251.075,-61.297,-176.868,6.372,148.231
C02812=1227.544,251.323,-61.324,-176.866,6.374,148.231
C02813=1227.540,251.572,-61.350,-176.864,6.376,148.230
C02814=1227.535,251.820,-61.377,-176.861,6.378,148.230
C02815=1227.531,252.069,-61.404,-176.858,6.380,148.230
C02816=1227.527,252.318,-61.430,-176.856,6.382,148.230
C02817=1227.522,252.566,-61.457,-176.854,6.384,148.229
C02818=1227.518,252.814,-61.484,-176.851,6.386,148.229
C02819=1227.513,253.063,-61.511,-176.849,6.388,148.229
C02820=1227.508,253.312,-61.537,-176.846,6.390,148.229
C02821=1227.504,253.560,-61.563,-176.844,6.392,148.228
C02822=1227.500,253.809,-61.590,-176.841,6.393,148.228
C02823=1227.496,254.057,-61.617,-176.839,6.396,148.228
C02824=1227.491,254.305,-61.644,-176.836,6.398,148.228
C02825=1227.486,254.555,-61.670,-176.833,6.400,148.227
C02826=1227.482,254.803,-61.697,-176.831,6.402,148.227
C02827=1227.478,255.051,-61.724,-176.828,6.404,148.227
C02828=1227.474,255.300,-61.751,-176.826,6.406,148.227
C02829=1227.470,255.549,-61.778,-176.823,6.408,148.226
C02830=1227.465,255.797,-61.805,-176.821,6.410,148.226
C02831=1227.460,256.046,-61.831,-176.818,6.412,148.226
C02832=1227.456,256.294,-61.858,-176.816,6.414,148.226
C02833=1227.452,256.543,-61.885,-176.814,6.416,148.226
C02834=1227.447,256.791,-61.912,-176.811,6.418,148.225
C02835=1227.442,257.040,-61.939,-176.808,6.420,148.225
C02836=1227.438,257.288,-61.965,-176.806,6.422,148.225
C02837=1227.434,257.537,-61.992,-176.804,6.424,148.225
C02838=1227.429,257.785,-62.019,-176.801,6.426,148.224
C02839=1227.424,258.034,-62.046,-176.799,6.428,148.224
C02840=1227.420,258.282,-62.073,-176.796,6.430,148.224
C02841=1227.416,258.530,-62.100,-176.793,6.433,148.224
C02842=1227.412,258.779,-62.127,-176.791,6.435,148.224
C02843=1227.407,259.028,-62.154,-176.789,6.437,148.223
C02844=1227.403,259.276,-62.181,-176.786,6.439,148.223
C02845=1227.398,259.525,-62.208,-176.783,6.441,148.223
C02846=1227.394,259.773,-62.235,-176.781,6.443,148.223
C02847=1227.389,260.022,-62.262,-176.779,6.445,148.222
C02848=1227.384,260.270,-62.289,-176.776,6.447,148.222
C02849=1227.380,260.519,-62.316,-176.774,6.449,148.222
C02850=1227.376,260.768,-62.343,-176.771,6.451,148.222
C02851=1227.372,261.016,-62.370,-176.769,6.453,148.221
C02852=1227.367,261.264,-62.397,-176.767,6.455,148.221
C02853=1227.363,261.513,-62.424,-176.763,6.458,148.221
C02854=1227.358,261.761,-62.452,-176.761,6.460,148.221
C02855=1227.354,262.009,-62.479,-176.759,6.462,148.221
C02856=1227.349,262.259,-62.507,-176.756,6.464,148.220
C02857=1227.346,262.507,-62.533,-176.754,6.466,148.220
C02858=1227.341,262.755,-62.560,-176.751,6.468,148.220
C02859=1227.336,263.004,-62.587,-176.749,6.470,148.220
C02860=1227.331,263.276,-62.617,-176.747,6.472,148.220
C02861=1227.326,263.549,-62.647,-176.743,6.474,148.219
C02862=1227.322,263.821,-62.677,-176.741,6.476,148.219
C02863=1227.317,264.094,-62.707,-176.738,6.479,148.219
C02864=1227.313,264.343,-62.735,-176.736,6.481,148.219
C02865=1227.308,264.591,-62.762,-176.733,6.483,148.218
C02866=1227.303,264.840,-62.789,-176.730,6.485,148.218
C02867=1227.299,265.088,-62.817,-176.728,6.487,148.218
C02868=1227.295,265.337,-62.844,-176.726,6.489,148.218
C02869=1227.290,265.585,-62.871,-176.723,6.491,148.218
C02870=1227.286,265.833,-62.899,-176.721,6.493,148.217
C02871=1227.281,266.082,-62.926,-176.718,6.496,148.217
C02872=1227.277,266.330,-62.953,-176.716,6.498,148.217
C02873=1227.273,266.579,-62.981,-176.713,6.500,148.217
C02874=1227.268,266.827,-63.008,-176.711,6.502,148.217
C02875=1227.263,267.076,-63.035,-176.708,6.504,148.216
C02876=1227.259,267.324,-63.063,-176.706,6.506,148.216
C02877=1227.255,267.573,-63.090,-176.704,6.508,148.216
C02878=1227.251,267.821,-63.118,-176.701,6.510,148.216
C02879=1227.246,268.069,-63.145,-176.698,6.513,148.216
C02880=1227.242,268.318,-63.173,-176.696,6.515,148.215
C02881=1227.238,268.566,-63.200,-176.694,6.517,148.215
C02882=1227.233,268.815,-63.227,-176.691,6.519,148.215
C02883=1227.229,269.063,-63.255,-176.688,6.521,148.215
C02884=1227.225,269.312,-63.283,-176.686,6.523,148.215
C02885=1227.220,269.560,-63.310,-176.684,6.525,148.214
C02886=1227.216,269.808,-63.338,-176.681,6.528,148.214
C02887=1227.211,270.057,-63.366,-176.678,6.530,148.214
C02888=1227.206,270.306,-63.393,-176.676,6.532,148.214
C02889=1227.202,270.553,-63.421,-176.674,6.534,148.214
C02890=1227.198,270.803,-63.449,-176.672,6.536,148.213
C02891=1227.194,271.051,-63.476,-176.669,6.538,148.213
C02892=1227.189,271.299,-63.503,-176.666,6.540,148.213
C02893=1227.185,271.548,-63.532,-176.664,6.543,148.213
C02894=1227.180,271.796,-63.559,-176.661,6.545,148.213
C02895=1227.176,272.044,-63.587,-176.659,6.547,148.212
C02896=1227.172,272.293,-63.615,-176.656,6.549,148.212
C02897=1227.167,272.541,-63.642,-176.654,6.552,148.212
C02898=1227.163,272.789,-63.670,-176.652,6.553,148.212
C02899=1227.158,273.038,-63.699,-176.650,6.556,148.212
C02900=1227.154,273.287,-63.726,-176.646,6.558,148.211
C02901=1227.149,273.535,-63.754,-176.644,6.561,148.211
C02902=1227.146,273.783,-63.782,-176.642,6.562,148.211
C02903=1227.141,274.032,-63.809,-176.640,6.565,148.211
C02904=1227.136,274.280,-63.837,-176.637,6.567,148.211
C02905=1227.132,274.528,-63.865,-176.635,6.569,148.211
C02906=1227.127,274.777,-63.892,-176.632,6.571,148.210
C02907=1227.124,275.025,-63.920,-176.630,6.574,148.210
C02908=1227.119,275.274,-63.949,-176.627,6.576,148.210
C02909=1227.115,275.522,-63.977,-176.625,6.578,148.210
C02910=1227.110,275.771,-64.004,-176.622,6.580,148.210
C02911=1227.106,276.019,-64.032,-176.620,6.583,148.210
C02912=1227.101,276.267,-64.061,-176.617,6.585,148.209
C02913=1227.097,276.515,-64.088,-176.615,6.587,148.209
C02914=1227.093,276.765,-64.116,-176.612,6.589,148.209
C02915=1227.088,277.013,-64.144,-176.610,6.591,148.209
C02916=1227.084,277.261,-64.172,-176.608,6.593,148.209
C02917=1227.080,277.509,-64.200,-176.605,6.596,148.209
C02918=1227.075,277.757,-64.228,-176.602,6.598,148.208
C02919=1227.071,278.006,-64.257,-176.600,6.600,148.208
C02920=1227.067,278.254,-64.284,-176.598,6.602,148.208
C02921=1227.062,278.503,-64.312,-176.595,6.604,148.208
C02922=1227.057,278.751,-64.340,-176.592,6.607,148.208
C02923=1227.054,279.000,-64.368,-176.590,6.609,148.208
C02924=1227.049,279.248,-64.397,-176.588,6.611,148.208
C02925=1227.045,279.497,-64.425,-176.585,6.613,148.207
C02926=1227.040,279.745,-64.453,-176.583,6.615,148.207
C02927=1227.036,279.993,-64.481,-176.580,6.618,148.207
C02928=1227.032,280.241,-64.509,-176.578,6.620,148.207
C02929=1227.027,280.490,-64.538,-176.575,6.622,148.207
C02930=1227.023,280.738,-64.566,-176.573,6.624,148.207
C02931=1227.018,280.987,-64.594,-176.571,6.626,148.206
C02932=1227.014,281.235,-64.622,-176.568,6.629,148.206
C02933=1227.009,281.484,-64.651,-176.566,6.632,148.206
C02934=1227.005,281.731,-64.679,-176.563,6.633,148.206
C02935=1227.001,281.980,-64.707,-176.561,6.636,148.206
C02936=1226.996,282.228,-64.735,-176.559,6.638,148.206
C02937=1226.993,282.477,-64.763,-176.556,6.641,148.205
C02938=1226.987,282.725,-64.792,-176.554,6.643,148.205
C02939=1226.984,282.974,-64.820,-176.551,6.645,148.205
C02940=1226.979,283.222,-64.848,-176.549,6.647,148.205
C02941=1226.975,283.470,-64.877,-176.547,6.649,148.205
C02942=1226.971,283.719,-64.906,-176.544,6.652,148.205
C02943=1226.966,283.967,-64.934,-176.542,6.654,148.205
C02944=1226.962,284.215,-64.962,-176.539,6.656,148.204
C02945=1226.957,284.464,-64.991,-176.537,6.658,148.204
C02946=1226.953,284.712,-65.019,-176.534,6.661,148.204
C02947=1226.948,284.960,-65.048,-176.532,6.663,148.204
C02948=1226.944,285.208,-65.076,-176.530,6.665,148.204
C02949=1226.940,285.457,-65.105,-176.527,6.667,148.204
C02950=1226.936,285.705,-65.133,-176.525,6.670,148.204
C02951=1226.931,285.954,-65.161,-176.522,6.673,148.204
C02952=1226.926,286.201,-65.190,-176.520,6.674,148.203
C02953=1226.923,286.450,-65.218,-176.518,6.677,148.203
C02954=1226.918,286.699,-65.247,-176.516,6.679,148.203
C02955=1226.914,286.947,-65.275,-176.512,6.682,148.203
C02956=1226.910,287.195,-65.304,-176.510,6.684,148.203
C02957=1226.904,287.443,-65.333,-176.508,6.686,148.203
C02958=1226.901,287.692,-65.361,-176.506,6.688,148.203
C02959=1226.897,287.940,-65.390,-176.503,6.691,148.203
C02960=1226.891,288.188,-65.419,-176.501,6.693,148.202
C02961=1226.888,288.437,-65.447,-176.498,6.695,148.202
C02962=1226.884,288.685,-65.476,-176.496,6.697,148.202
C02963=1226.878,288.933,-65.505,-176.493,6.700,148.202
C02964=1226.874,289.208,-65.536,-176.491,6.702,148.202
C02965=1226.870,289.482,-65.567,-176.488,6.705,148.202
C02966=1226.865,289.755,-65.600,-176.486,6.707,148.202
C02967=1226.860,290.030,-65.631,-176.483,6.710,148.201
C02968=1226.855,290.278,-65.660,-176.480,6.712,148.201
C02969=1226.851,290.526,-65.689,-176.478,6.714,148.201
C02970=1226.846,290.775,-65.718,-176.476,6.717,148.201
C02971=1226.842,291.022,-65.746,-176.473,6.720,148.201
C02972=1226.838,291.271,-65.775,-176.471,6.722,148.201
C02973=1226.834,291.520,-65.805,-176.469,6.724,148.201
C02974=1226.829,291.768,-65.833,-176.466,6.727,148.201
C02975=1226.825,292.016,-65.862,-176.464,6.729,148.200
C02976=1226.821,292.265,-65.891,-176.461,6.731,148.200
C02977=1226.816,292.512,-65.920,-176.459,6.734,148.200
C02978=1226.811,292.761,-65.948,-176.457,6.736,148.200
C02979=1226.808,293.009,-65.977,-176.454,6.738,148.200
C02980=1226.804,293.258,-66.006,-176.452,6.740,148.200
C02981=1226.799,293.505,-66.035,-176.449,6.743,148.200
C02982=1226.794,293.754,-66.064,-176.447,6.746,148.200
C02983=1226.790,294.003,-66.093,-176.445,6.748,148.200
C02984=1226.787,294.251,-66.122,-176.442,6.750,148.200
C02985=1226.782,294.499,-66.151,-176.440,6.753,148.200
C02986=1226.777,294.747,-66.180,-176.438,6.755,148.199
C02987=1226.773,294.995,-66.209,-176.435,6.757,148.199
C02988=1226.769,295.244,-66.238,-176.433,6.759,148.199
C02989=1226.764,295.492,-66.267,-176.430,6.762,148.199
C02990=1226.760,295.740,-66.297,-176.428,6.764,148.199
C02991=1226.756,295.989,-66.325,-176.426,6.767,148.199
C02992=1226.752,296.237,-66.354,-176.423,6.769,148.199
C02993=1226.748,296.485,-66.384,-176.421,6.772,148.199
C02994=1226.743,296.733,-66.412,-176.419,6.774,148.199
C02995=1226.738,296.982,-66.442,-176.417,6.776,148.199
C02996=1226.734,297.230,-66.471,-176.414,6.779,148.199
C02997=1226.730,297.478,-66.501,-176.411,6.781,148.198
C02998=1226.726,297.727,-66.529,-176.409,6.783,148.198
C02999=1226.721,297.975,-66.558,-176.407,6.786,148.198
C03000=1226.717,298.223,-66.588,-176.405,6.788,148.198
C03001=1226.712,298.471,-66.617,-176.402,6.791,148.198
C03002=1226.708,298.719,-66.647,-176.400,6.793,148.198
C03003=1226.704,298.968,-66.675,-176.397,6.796,148.198
C03004=1226.699,299.216,-66.705,-176.395,6.798,148.198
C03005=1226.695,299.464,-66.734,-176.393,6.800,148.198
C03006=1226.691,299.712,-66.763,-176.390,6.803,148.198
C03007=1226.686,299.961,-66.793,-176.388,6.805,148.198
C03008=1226.682,300.209,-66.822,-176.386,6.808,148.198
C03009=1226.678,300.457,-66.852,-176.383,6.809,148.197
C03010=1226.674,300.705,-66.881,-176.381,6.813,148.197
C03011=1226.669,300.953,-66.910,-176.379,6.815,148.197
C03012=1226.665,301.202,-66.939,-176.377,6.817,148.197
C03013=1226.660,301.450,-66.969,-176.374,6.820,148.197
C03014=1226.656,301.698,-66.998,-176.372,6.822,148.197
C03015=1226.652,301.947,-67.027,-176.370,6.824,148.197
C03016=1226.648,302.195,-67.057,-176.367,6.828,148.197
C03017=1226.644,302.443,-67.086,-176.364,6.829,148.197
C03018=1226.639,302.692,-67.116,-176.362,6.832,148.197
C03019=1226.635,302.939,-67.145,-176.360,6.835,148.197
C03020=1226.631,303.187,-67.174,-176.358,6.837,148.197
C03021=1226.626,303.436,-67.204,-176.356,6.839,148.197
C03022=1226.621,303.684,-67.234,-176.353,6.841,148.197
C03023=1226.617,303.932,-67.263,-176.351,6.844,148.197
C03024=1226.613,304.181,-67.293,-176.349,6.847,148.196
C03025=1226.609,304.428,-67.323,-176.347,6.849,148.196
C03026=1226.605,304.677,-67.352,-176.344,6.852,148.196
C03027=1226.601,304.925,-67.382,-176.342,6.854,148.196
C03028=1226.597,305.173,-67.411,-176.340,6.856,148.196
C03029=1226.592,305.422,-67.441,-176.337,6.859,148.196
C03030=1226.588,305.670,-67.471,-176.334,6.861,148.196
C03031=1226.583,305.918,-67.500,-176.332,6.863,148.196
C03032=1226.579,306.167,-67.530,-176.330,6.867,148.196
C03033=1226.575,306.413,-67.560,-176.328,6.869,148.196
C03034=1226.570,306.662,-67.590,-176.325,6.871,148.196
C03035=1226.566,306.910,-67.619,-176.323,6.874,148.196
C03036=1226.561,307.159,-67.648,-176.321,6.876,148.196
C03037=1226.557,307.407,-67.678,-176.319,6.878,148.196
C03038=1226.553,307.655,-67.709,-176.316,6.881,148.196
C03039=1226.548,307.903,-67.738,-176.314,6.884,148.196
C03040=1226.544,308.151,-67.768,-176.312,6.886,148.196
C03041=1226.540,308.400,-67.797,-176.310,6.888,148.196
C03042=1226.535,308.648,-67.828,-176.307,6.891,148.196
C03043=1226.531,308.896,-67.857,-176.305,6.893,148.196
C03044=1226.527,309.144,-67.887,-176.303,6.896,148.195
C03045=1226.523,309.392,-67.917,-176.300,6.899,148.195
C03046=1226.518,309.640,-67.947,-176.298,6.901,148.195
C03047=1226.514,309.889,-67.976,-176.296,6.903,148.195
C03048=1226.510,310.137,-68.006,-176.293,6.906,148.195
C03049=1226.505,310.385,-68.037,-176.291,6.908,148.195
C03050=1226.501,310.633,-68.066,-176.289,6.911,148.195
C03051=1226.498,310.881,-68.097,-176.286,6.914,148.195
C03052=1226.493,311.130,-68.127,-176.285,6.916,148.195
C03053=1226.489,311.378,-68.156,-176.283,6.918,148.195
C03054=1226.485,311.626,-68.186,-176.280,6.922,148.195
C03055=1226.480,311.875,-68.216,-176.278,6.924,148.195
C03056=1226.476,312.122,-68.246,-176.276,6.926,148.195
C03057=1226.472,312.370,-68.276,-176.273,6.929,148.195
C03058=1226.467,312.618,-68.307,-176.271,6.931,148.195
C03059=1226.463,312.867,-68.336,-176.269,6.933,148.195
C03060=1226.458,313.115,-68.366,-176.266,6.937,148.195
C03061=1226.454,313.363,-68.396,-176.264,6.939,148.195
C03062=1226.450,313.611,-68.426,-176.262,6.941,148.195
C03063=1226.446,313.859,-68.457,-176.259,6.944,148.195
C03064=1226.441,314.107,-68.486,-176.258,6.947,148.195
C03065=1226.437,314.356,-68.517,-176.256,6.949,148.195
C03066=1226.433,314.604,-68.547,-176.253,6.952,148.195
C03067=1226.429,314.852,-68.577,-176.251,6.954,148.195
C03068=1226.425,315.128,-68.611,-176.248,6.957,148.195
C03069=1226.419,315.403,-68.644,-176.246,6.959,148.195
C03070=1226.415,315.679,-68.678,-176.243,6.962,148.195
C03071=1226.410,315.955,-68.712,-176.241,6.965,148.195
C03072=1226.406,316.203,-68.742,-176.239,6.968,148.195
C03073=1226.401,316.452,-68.772,-176.236,6.971,148.195
C03074=1226.397,316.699,-68.802,-176.234,6.973,148.195
C03075=1226.392,316.947,-68.833,-176.232,6.975,148.195
C03076=1226.389,317.196,-68.862,-176.230,6.979,148.195
C03077=1226.384,317.444,-68.893,-176.228,6.981,148.195
C03078=1226.380,317.692,-68.923,-176.225,6.983,148.195
C03079=1226.375,317.940,-68.953,-176.223,6.986,148.195
C03080=1226.372,318.188,-68.984,-176.221,6.989,148.195
C03081=1226.367,318.436,-69.014,-176.219,6.991,148.195
C03082=1226.363,318.685,-69.046,-176.216,6.994,148.195
C03083=1226.359,318.933,-69.075,-176.214,6.996,148.195
C03084=1226.354,319.181,-69.106,-176.212,6.998,148.195
C03085=1226.350,319.428,-69.136,-176.210,7.002,148.195
C03086=1226.346,319.676,-69.167,-176.208,7.004,148.195
C03087=1226.342,319.925,-69.197,-176.206,7.006,148.195
C03088=1226.337,320.173,-69.227,-176.203,7.009,148.195
C03089=1226.333,320.421,-69.258,-176.202,7.012,148.195
C03090=1226.329,320.669,-69.288,-176.199,7.014,148.195
C03091=1226.324,320.917,-69.319,-176.197,7.017,148.195
C03092=1226.321,321.165,-69.349,-176.195,7.019,148.195
C03093=1226.316,321.414,-69.380,-176.193,7.022,148.196
C03094=1226.312,321.662,-69.410,-176.190,7.025,148.196
C03095=1226.308,321.909,-69.440,-176.188,7.027,148.195
C03096=1226.304,322.158,-69.472,-176.186,7.029,148.195
C03097=1226.299,322.406,-69.502,-176.184,7.033,148.196
C03098=1226.295,322.654,-69.533,-176.182,7.035,148.196
C03099=1226.291,322.902,-69.563,-176.180,7.037,148.196
C03100=1226.287,323.150,-69.594,-176.178,7.040,148.196
C03101=1226.283,323.398,-69.625,-176.176,7.043,148.196
C03102=1226.278,323.646,-69.655,-176.173,7.045,148.196
C03103=1226.273,323.894,-69.686,-176.171,7.048,148.196
C03104=1226.269,324.143,-69.717,-176.169,7.050,148.196
C03105=1226.266,324.390,-69.747,-176.166,7.053,148.196
C03106=1226.261,324.638,-69.778,-176.165,7.056,148.196
C03107=1226.257,324.887,-69.809,-176.163,7.058,148.196
C03108=1226.253,325.134,-69.839,-176.160,7.061,148.196
C03109=1226.248,325.382,-69.870,-176.158,7.064,148.196
C03110=1226.244,325.630,-69.901,-176.156,7.066,148.196
C03111=1226.240,325.879,-69.932,-176.154,7.069,148.196
C03112=1226.235,326.127,-69.963,-176.152,7.072,148.196
C03113=1226.231,326.375,-69.993,-176.150,7.074,148.196
C03114=1226.227,326.623,-70.024,-176.148,7.077,148.197
C03115=1226.223,326.871,-70.055,-176.146,7.079,148.196
C03116=1226.218,327.119,-70.086,-176.144,7.082,148.196
C03117=1226.215,327.368,-70.116,-176.141,7.085,148.197
C03118=1226.211,327.615,-70.148,-176.139,7.087,148.197
C03119=1226.206,327.863,-70.179,-176.138,7.090,148.197
C03120=1226.202,328.112,-70.210,-176.135,7.093,148.197
C03121=1226.197,328.359,-70.240,-176.133,7.095,148.197
C03122=1226.193,328.607,-70.271,-176.131,7.098,148.197
C03123=1226.189,328.856,-70.302,-176.129,7.101,148.197
C03124=1226.185,329.103,-70.333,-176.127,7.103,148.197
C03125=1226.180,329.351,-70.364,-176.125,7.105,148.197
C03126=1226.176,329.600,-70.395,-176.123,7.109,148.197
C03127=1226.172,329.848,-70.426,-176.121,7.111,148.197
C03128=1226.168,330.096,-70.457,-176.119,7.114,148.197
C03129=1226.164,330.344,-70.488,-176.116,7.117,148.197
C03130=1226.159,330.592,-70.519,-176.114,7.119,148.197
C03131=1226.155,330.840,-70.550,-176.113,7.121,148.198
C03132=1226.151,331.088,-70.582,-176.110,7.124,148.198
C03133=1226.147,331.336,-70.612,-176.108,7.127,148.198
C03134=1226.143,331.584,-70.643,-176.106,7.129,148.198
C03135=1226.138,331.831,-70.675,-176.104,7.133,148.198
C03136=1226.134,332.080,-70.706,-176.102,7.135,148.198
C03137=1226.130,332.328,-70.736,-176.100,7.137,148.198
C03138=1226.126,332.576,-70.768,-176.098,7.141,148.198
C03139=1226.121,332.824,-70.799,-176.096,7.143,148.198
C03140=1226.117,333.072,-70.830,-176.094,7.145,148.198
C03141=1226.113,333.320,-70.862,-176.092,7.148,148.198
C03142=1226.109,333.568,-70.892,-176.090,7.151,148.199
C03143=1226.105,333.816,-70.924,-176.088,7.153,148.199
C03144=1226.100,334.064,-70.955,-176.086,7.157,148.199
C03145=1226.096,334.313,-70.986,-176.084,7.159,148.199
C03146=1226.092,334.560,-71.018,-176.082,7.161,148.199
C03147=1226.088,334.808,-71.049,-176.080,7.165,148.199
C03148=1226.084,335.056,-71.080,-176.078,7.167,148.199
C03149=1226.079,335.304,-71.111,-176.076,7.169,148.199
C03150=1226.075,335.552,-71.143,-176.074,7.172,148.199
C03151=1226.071,335.800,-71.174,-176.072,7.175,148.200
C03152=1226.067,336.048,-71.206,-176.070,7.178,148.200
C03153=1226.062,336.296,-71.237,-176.068,7.181,148.200
C03154=1226.058,336.544,-71.269,-176.066,7.183,148.200
C03155=1226.053,336.792,-71.299,-176.064,7.185,148.200
C03156=1226.050,337.040,-71.331,-176.062,7.189,148.200
C03157=1226.045,337.287,-71.363,-176.060,7.191,148.200
C03158=1226.041,337.536,-71.394,-176.058,7.193,148.200
C03159=1226.037,337.783,-71.425,-176.056,7.197,148.200
C03160=1226.033,338.032,-71.457,-176.054,7.199,148.201
C03161=1226.029,338.279,-71.488,-176.052,7.202,148.201
C03162=1226.025,338.527,-71.520,-176.050,7.205,148.201
C03163=1226.020,338.776,-71.551,-176.048,7.207,148.201
C03164=1226.016,339.024,-71.583,-176.047,7.210,148.201
C03165=1226.011,339.272,-71.614,-176.044,7.213,148.201
C03166=1226.007,339.520,-71.646,-176.042,7.216,148.201
C03167=1226.004,339.768,-71.678,-176.041,7.218,148.202
C03168=1225.999,340.016,-71.708,-176.038,7.221,148.202
C03169=1225.995,340.264,-71.741,-176.037,7.224,148.202
C03170=1225.990,340.511,-71.772,-176.035,7.226,148.202
C03171=1225.987,340.760,-71.804,-176.033,7.229,148.202
C03172=1225.982,341.038,-71.839,-176.031,7.232,148.202
C03173=1225.977,341.314,-71.874,-176.028,7.235,148.202
C03174=1225.972,341.592,-71.910,-176.026,7.239,148.203
C03175=1225.967,341.870,-71.945,-176.024,7.241,148.203
C03176=1225.964,342.119,-71.977,-176.022,7.244,148.203
C03177=1225.959,342.366,-72.009,-176.020,7.247,148.203
C03178=1225.955,342.614,-72.041,-176.019,7.249,148.203
C03179=1225.950,342.862,-72.072,-176.017,7.253,148.203
C03180=1225.947,343.110,-72.104,-176.014,7.255,148.203
C03181=1225.942,343.358,-72.135,-176.013,7.257,148.204
C03182=1225.938,343.606,-72.168,-176.011,7.260,148.204
C03183=1225.934,343.854,-72.199,-176.009,7.263,148.204
C03184=1225.930,344.101,-72.231,-176.007,7.266,148.204
C03185=1225.925,344.350,-72.263,-176.006,7.268,148.204
C03186=1225.921,344.598,-72.294,-176.003,7.271,148.204
C03187=1225.917,344.846,-72.326,-176.001,7.274,148.204
C03188=1225.913,345.094,-72.358,-176.000,7.276,148.205
C03189=1225.908,345.341,-72.390,-175.998,7.279,148.205
C03190=1225.905,345.589,-72.422,-175.996,7.282,148.205
C03191=1225.900,345.838,-72.454,-175.994,7.285,148.205
C03192=1225.896,346.085,-72.486,-175.993,7.287,148.205
C03193=1225.892,346.333,-72.517,-175.991,7.291,148.206
C03194=1225.888,346.581,-72.550,-175.989,7.293,148.206
C03195=1225.884,346.829,-72.581,-175.987,7.295,148.206
C03196=1225.880,347.077,-72.613,-175.985,7.298,148.206
C03197=1225.875,347.324,-72.645,-175.983,7.301,148.206
C03198=1225.871,347.572,-72.677,-175.981,7.304,148.206
C03199=1225.867,347.821,-72.709,-175.980,7.306,148.207
C03200=1225.862,348.068,-72.741,-175.978,7.310,148.207
C03201=1225.859,348.316,-72.773,-175.976,7.312,148.207
C03202=1225.854,348.565,-72.805,-175.974,7.315,148.207
C03203=1225.850,348.813,-72.837,-175.973,7.317,148.207
C03204=1225.845,349.060,-72.869,-175.971,7.321,148.208
C03205=1225.842,349.308,-72.901,-175.969,7.323,148.208
C03206=1225.838,349.556,-72.933,-175.967,7.326,148.208
C03207=1225.833,349.804,-72.965,-175.966,7.328,148.208
C03208=1225.829,350.052,-72.997,-175.963,7.332,148.208
C03209=1225.825,350.300,-73.030,-175.962,7.334,148.209
C03210=1225.821,350.547,-73.062,-175.960,7.337,148.209
C03211=1225.816,350.795,-73.094,-175.958,7.340,148.209
C03212=1225.813,351.043,-73.126,-175.956,7.343,148.209
C03213=1225.808,351.292,-73.158,-175.955,7.345,148.209
C03214=1225.804,351.539,-73.190,-175.953,7.348,148.210
C03215=1225.800,351.787,-73.223,-175.951,7.351,148.210
C03216=1225.796,352.035,-73.255,-175.949,7.354,148.210
C03217=1225.792,352.283,-73.287,-175.948,7.356,148.210
C03218=1225.787,352.531,-73.319,-175.947,7.359,148.211
C03219=1225.783,352.779,-73.351,-175.944,7.362,148.211
C03220=1225.779,353.026,-73.384,-175.943,7.365,148.211
C03221=1225.775,353.275,-73.416,-175.941,7.367,148.211
C03222=1225.771,353.522,-73.448,-175.939,7.370,148.211
C03223=1225.766,353.770,-73.480,-175.937,7.373,148.212
C03224=1225.763,354.018,-73.513,-175.936,7.376,148.212
C03225=1225.758,354.266,-73.545,-175.934,7.378,148.212
C03226=1225.753,354.514,-73.577,-175.932,7.381,148.212
C03227=1225.750,354.761,-73.610,-175.931,7.384,148.212
C03228=1225.746,355.010,-73.642,-175.929,7.387,148.213
C03229=1225.742,355.258,-73.674,-175.927,7.390,148.213
C03230=1225.737,355.505,-73.707,-175.926,7.392,148.213
C03231=1225.733,355.753,-73.739,-175.924,7.395,148.213
C03232=1225.729,356.001,-73.771,-175.922,7.398,148.214
C03233=1225.725,356.249,-73.804,-175.921,7.401,148.214
C03234=1225.721,356.497,-73.836,-175.919,7.403,148.214
C03235=1225.716,356.744,-73.869,-175.918,7.406,148.214
C03236=1225.712,356.992,-73.901,-175.916,7.408,148.214
C03237=1225.708,357.240,-73.933,-175.914,7.412,148.215
C03238=1225.704,357.488,-73.966,-175.913,7.415,148.215
C03239=1225.700,357.736,-73.998,-175.911,7.417,148.215
C03240=1225.696,357.984,-74.031,-175.909,7.420,148.215
C03241=1225.691,358.231,-74.063,-175.908,7.422,148.216
C03242=1225.688,358.479,-74.096,-175.906,7.426,148.216
C03243=1225.683,358.727,-74.128,-175.904,7.428,148.216
C03244=1225.679,358.975,-74.162,-175.903,7.431,148.216
C03245=1225.675,359.223,-74.193,-175.902,7.434,148.217
C03246=1225.671,359.471,-74.227,-175.900,7.436,148.217
C03247=1225.667,359.719,-74.259,-175.898,7.440,148.217
C03248=1225.662,359.966,-74.292,-175.897,7.442,148.218
C03249=1225.658,360.214,-74.324,-175.895,7.445,148.218
C03250=1225.654,360.462,-74.357,-175.893,7.447,148.218
C03251=1225.650,360.710,-74.389,-175.892,7.450,148.218
C03252=1225.646,360.958,-74.422,-175.890,7.453,148.219
C03253=1225.642,361.206,-74.454,-175.888,7.456,148.219
C03254=1225.638,361.454,-74.487,-175.887,7.459,148.219
C03255=1225.634,361.701,-74.520,-175.886,7.462,148.219
C03256=1225.629,361.949,-74.552,-175.884,7.464,148.220
C03257=1225.625,362.196,-74.585,-175.883,7.467,148.220
C03258=1225.621,362.445,-74.618,-175.881,7.469,148.220
C03259=1225.617,362.693,-74.651,-175.879,7.473,148.221
C03260=1225.613,362.940,-74.683,-175.878,7.476,148.221
C03261=1225.609,363.188,-74.716,-175.877,7.478,148.221
C03262=1225.605,363.436,-74.749,-175.875,7.481,148.221
C03263=1225.601,363.684,-74.782,-175.874,7.484,148.222
C03264=1225.596,363.932,-74.814,-175.872,7.486,148.222
C03265=1225.593,364.180,-74.847,-175.871,7.489,148.222
C03266=1225.589,364.427,-74.880,-175.869,7.492,148.223
C03267=1225.584,364.675,-74.912,-175.867,7.495,148.223
C03268=1225.579,364.923,-74.945,-175.866,7.498,148.223
C03269=1225.575,365.170,-74.979,-175.864,7.500,148.223
C03270=1225.571,365.418,-75.012,-175.863,7.503,148.224
C03271=1225.567,365.666,-75.044,-175.862,7.506,148.224
C03272=1225.563,365.914,-75.077,-175.860,7.509,148.224
C03273=1225.559,366.162,-75.110,-175.859,7.511,148.225
C03274=1225.555,366.409,-75.143,-175.858,7.514,148.225
C03275=1225.551,366.658,-75.175,-175.856,7.517,148.225
C03276=1225.546,366.937,-75.213,-175.854,7.520,148.226
C03277=1225.541,367.217,-75.251,-175.853,7.523,148.226
C03278=1225.537,367.497,-75.287,-175.851,7.526,148.226
C03279=1225.533,367.776,-75.324,-175.850,7.529,148.227
C03280=1225.528,368.024,-75.357,-175.849,7.532,148.227
C03281=1225.524,368.272,-75.391,-175.847,7.534,148.227
C03282=1225.520,368.519,-75.424,-175.846,7.537,148.228
C03283=1225.516,368.767,-75.457,-175.845,7.540,148.228
C03284=1225.512,369.016,-75.489,-175.842,7.543,148.228
C03285=1225.508,369.263,-75.523,-175.841,7.546,148.229
C03286=1225.503,369.511,-75.556,-175.840,7.549,148.229
C03287=1225.499,369.759,-75.589,-175.838,7.552,148.229
C03288=1225.495,370.006,-75.622,-175.837,7.554,148.230
C03289=1225.491,370.254,-75.655,-175.836,7.557,148.230
C03290=1225.487,370.502,-75.688,-175.834,7.560,148.230
C03291=1225.483,370.750,-75.721,-175.833,7.563,148.231
C03292=1225.479,370.997,-75.755,-175.832,7.565,148.231
C03293=1225.474,371.245,-75.788,-175.830,7.568,148.231
C03294=1225.470,371.493,-75.821,-175.829,7.571,148.232
C03295=1225.466,371.741,-75.854,-175.828,7.574,148.232
C03296=1225.462,371.988,-75.887,-175.827,7.576,148.232
C03297=1225.458,372.236,-75.920,-175.825,7.579,148.233
C03298=1225.454,372.484,-75.954,-175.824,7.582,148.233
C03299=1225.450,372.732,-75.987,-175.823,7.585,148.233
C03300=1225.445,372.979,-76.020,-175.821,7.587,148.234
C03301=1225.441,373.227,-76.053,-175.820,7.590,148.234
C03302=1225.437,373.475,-76.086,-175.819,7.593,148.234
C03303=1225.433,373.722,-76.119,-175.818,7.595,148.235
C03304=1225.429,373.970,-76.152,-175.817,7.598,148.235
C03305=1225.425,374.218,-76.186,-175.816,7.600,148.235
C03306=1225.421,374.466,-76.219,-175.814,7.603,148.236
C03307=1225.416,374.713,-76.252,-175.813,7.606,148.236
C03308=1225.412,374.961,-76.285,-175.812,7.609,148.236
C03309=1225.408,375.209,-76.318,-175.811,7.611,148.237
C03310=1225.404,375.457,-76.351,-175.810,7.614,148.237
C03311=1225.401,375.705,-76.385,-175.808,7.617,148.237
C03312=1225.397,375.952,-76.419,-175.807,7.620,148.238
C03313=1225.393,376.200,-76.452,-175.806,7.622,148.238
C03314=1225.388,376.448,-76.485,-175.805,7.625,148.239
C03315=1225.384,376.696,-76.519,-175.803,7.628,148.239
C03316=1225.379,376.943,-76.552,-175.803,7.630,148.239
C03317=1225.375,377.191,-76.585,-175.802,7.633,148.240
C03318=1225.371,377.438,-76.619,-175.800,7.636,148.240
C03319=1225.367,377.686,-76.652,-175.799,7.638,148.240
C03320=1225.363,377.934,-76.685,-175.798,7.641,148.241
C03321=1225.359,378.181,-76.719,-175.796,7.644,148.241
C03322=1225.355,378.430,-76.752,-175.795,7.647,148.242
C03323=1225.351,378.677,-76.787,-175.795,7.649,148.242
C03324=1225.347,378.925,-76.820,-175.793,7.651,148.242
C03325=1225.343,379.173,-76.853,-175.792,7.654,148.243
C03326=1225.338,379.420,-76.886,-175.791,7.657,148.243
C03327=1225.334,379.668,-76.919,-175.790,7.660,148.244
C03328=1225.331,379.915,-76.953,-175.789,7.663,148.244
C03329=1225.326,380.163,-76.987,-175.788,7.665,148.244
C03330=1225.322,380.412,-77.020,-175.787,7.668,148.245
C03331=1225.318,380.659,-77.054,-175.786,7.670,148.245
C03332=1225.314,380.907,-77.087,-175.785,7.673,148.245
C03333=1225.310,381.154,-77.120,-175.783,7.676,148.246
C03334=1225.305,381.402,-77.154,-175.783,7.678,148.246
C03335=1225.301,381.649,-77.188,-175.782,7.681,148.247
C03336=1225.297,381.897,-77.221,-175.780,7.684,148.247
C03337=1225.294,382.146,-77.255,-175.779,7.686,148.247
C03338=1225.290,382.393,-77.289,-175.778,7.689,148.248
C03339=1225.285,382.641,-77.322,-175.778,7.691,148.248
C03340=1225.281,382.888,-77.356,-175.776,7.694,148.249
C03341=1225.277,383.136,-77.389,-175.775,7.697,148.249
C03342=1225.273,383.383,-77.423,-175.774,7.700,148.249
C03343=1225.269,383.631,-77.457,-175.773,7.702,148.250
C03344=1225.265,383.879,-77.491,-175.772,7.705,148.250
C03345=1225.261,384.127,-77.524,-175.771,7.707,148.250
C03346=1225.257,384.374,-77.558,-175.770,7.709,148.251
C03347=1225.252,384.622,-77.591,-175.770,7.712,148.251
C03348=1225.249,384.870,-77.626,-175.768,7.715,148.252
C03349=1225.244,385.118,-77.659,-175.767,7.718,148.252
C03350=1225.240,385.366,-77.692,-175.767,7.720,148.253
C03351=1225.236,385.613,-77.726,-175.766,7.723,148.253
C03352=1225.232,385.860,-77.759,-175.764,7.726,148.253
C03353=1225.228,386.108,-77.794,-175.764,7.728,148.254
C03354=1225.224,386.356,-77.827,-175.763,7.730,148.254
C03355=1225.220,386.603,-77.861,-175.761,7.733,148.254
C03356=1225.216,386.851,-77.895,-175.761,7.736,148.255
C03357=1225.211,387.099,-77.929,-175.760,7.738,148.255
C03358=1225.207,387.347,-77.962,-175.759,7.741,148.256
C03359=1225.204,387.594,-77.996,-175.758,7.743,148.256
C03360=1225.199,387.842,-78.030,-175.757,7.746,148.257
C03361=1225.195,388.089,-78.064,-175.756,7.749,148.257
C03362=1225.191,388.337,-78.097,-175.755,7.751,148.257
C03363=1225.187,388.585,-78.132,-175.755,7.754,148.258
C03364=1225.183,388.833,-78.165,-175.753,7.757,148.258
C03365=1225.179,389.080,-78.199,-175.753,7.759,148.259
C03366=1225.174,389.328,-78.233,-175.752,7.762,148.259
C03367=1225.171,389.576,-78.267,-175.751,7.764,148.259
C03368=1225.166,389.823,-78.301,-175.750,7.767,148.260
C03369=1225.162,390.071,-78.335,-175.749,7.769,148.260
C03370=1225.158,390.318,-78.368,-175.748,7.771,148.261
C03371=1225.154,390.567,-78.403,-175.747,7.774,148.261
C03372=1225.150,390.814,-78.436,-175.747,7.776,148.261
C03373=1225.146,391.061,-78.470,-175.746,7.779,148.262
C03374=1225.141,391.309,-78.504,-175.745,7.782,148.262
C03375=1225.138,391.557,-78.538,-175.744,7.784,148.263
C03376=1225.133,391.805,-78.572,-175.743,7.787,148.263
C03377=1225.129,392.052,-78.606,-175.742,7.789,148.264
C03378=1225.126,392.300,-78.640,-175.741,7.792,148.264
C03379=1225.121,392.548,-78.674,-175.741,7.794,148.264
C03380=1225.117,392.829,-78.713,-175.740,7.797,148.265
C03381=1225.112,393.110,-78.751,-175.739,7.800,148.265
C03382=1225.107,393.392,-78.790,-175.738,7.803,148.266
C03383=1225.103,393.673,-78.829,-175.737,7.806,148.266
C03384=1225.098,393.921,-78.863,-175.736,7.808,148.267
C03385=1225.095,394.169,-78.897,-175.735,7.811,148.267
C03386=1225.091,394.416,-78.931,-175.735,7.813,148.268
C03387=1225.086,394.664,-78.965,-175.734,7.816,148.268
C03388=1225.082,394.911,-78.998,-175.733,7.818,148.269
C03389=1225.079,395.160,-79.033,-175.732,7.821,148.269
C03390=1225.075,395.407,-79.067,-175.731,7.823,148.269
C03391=1225.070,395.655,-79.101,-175.731,7.826,148.270
C03392=1225.067,395.903,-79.135,-175.730,7.828,148.270
C03393=1225.062,396.150,-79.170,-175.729,7.831,148.271
C03394=1225.058,396.397,-79.203,-175.729,7.833,148.271
C03395=1225.054,396.646,-79.238,-175.728,7.836,148.272
C03396=1225.050,396.893,-79.271,-175.727,7.838,148.272
C03397=1225.045,397.140,-79.306,-175.726,7.840,148.272
C03398=1225.042,397.388,-79.340,-175.726,7.843,148.273
C03399=1225.037,397.636,-79.374,-175.725,7.845,148.273
C03400=1225.034,397.883,-79.408,-175.724,7.847,148.274
C03401=1225.030,398.131,-79.443,-175.724,7.850,148.274
C03402=1225.026,398.379,-79.476,-175.722,7.853,148.275
C03403=1225.021,398.626,-79.511,-175.722,7.855,148.275
C03404=1225.018,398.874,-79.545,-175.722,7.857,148.275
C03405=1225.013,399.122,-79.579,-175.720,7.860,148.276
C03406=1225.008,399.369,-79.613,-175.720,7.862,148.276
C03407=1225.005,399.617,-79.648,-175.719,7.864,148.277
C03408=1225.001,399.864,-79.682,-175.718,7.867,148.277
C03409=1224.997,400.112,-79.716,-175.718,7.869,148.277
C03410=1224.993,400.360,-79.751,-175.717,7.872,148.278
C03411=1224.989,400.607,-79.785,-175.716,7.874,148.278
C03412=1224.984,400.855,-79.818,-175.716,7.876,148.279
C03413=1224.981,401.103,-79.853,-175.715,7.879,148.279
C03414=1224.976,401.350,-79.887,-175.714,7.881,148.280
C03415=1224.972,401.597,-79.922,-175.714,7.883,148.280
C03416=1224.969,401.845,-79.956,-175.713,7.886,148.280
C03417=1224.964,402.093,-79.990,-175.712,7.888,148.281
C03418=1224.961,402.340,-80.024,-175.712,7.890,148.281
C03419=1224.956,402.588,-80.059,-175.711,7.893,148.282
C03420=1224.952,402.835,-80.093,-175.710,7.895,148.282
C03421=1224.948,403.083,-80.128,-175.710,7.897,148.283
C03422=1224.944,403.331,-80.162,-175.709,7.900,148.283
C03423=1224.940,403.578,-80.195,-175.708,7.902,148.283
C03424=1224.936,403.826,-80.230,-175.708,7.904,148.284
C03425=1224.931,404.074,-80.265,-175.707,7.907,148.284
C03426=1224.928,404.322,-80.299,-175.706,7.909,148.285
C03427=1224.923,404.569,-80.333,-175.706,7.911,148.285
C03428=1224.920,404.816,-80.367,-175.706,7.913,148.286
C03429=1224.916,405.064,-80.402,-175.704,7.916,148.286
C03430=1224.911,405.312,-80.436,-175.704,7.918,148.286
C03431=1224.908,405.560,-80.471,-175.704,7.920,148.287
C03432=1224.903,405.807,-80.505,-175.702,7.923,148.287
C03433=1224.899,406.054,-80.540,-175.702,7.925,148.288
C03434=1224.895,406.302,-80.574,-175.702,7.928,148.288
C03435=1224.891,406.550,-80.608,-175.701,7.930,148.289
C03436=1224.887,406.798,-80.643,-175.700,7.932,148.289
C03437=1224.883,407.045,-80.677,-175.700,7.935,148.290
C03438=1224.878,407.292,-80.711,-175.699,7.937,148.290
C03439=1224.875,407.540,-80.747,-175.698,7.939,148.290
C03440=1224.871,407.787,-80.781,-175.698,7.941,148.291
C03441=1224.867,408.035,-80.816,-175.697,7.944,148.291
C03442=1224.862,408.282,-80.850,-175.696,7.946,148.291
C03443=1224.859,408.530,-80.884,-175.696,7.948,148.292
C03444=1224.855,408.778,-80.919,-175.696,7.950,148.292
C03445=1224.850,409.025,-80.953,-175.695,7.953,148.293
C03446=1224.847,409.273,-80.988,-175.694,7.955,148.293
C03447=1224.842,409.520,-81.022,-175.694,7.957,148.294
C03448=1224.838,409.768,-81.057,-175.693,7.959,148.294
C03449=1224.834,410.015,-81.091,-175.693,7.961,148.295
C03450=1224.830,410.264,-81.126,-175.692,7.963,148.295
C03451=1224.826,410.510,-81.161,-175.691,7.966,148.295
C03452=1224.822,410.759,-81.196,-175.691,7.968,148.296
C03453=1224.818,411.006,-81.230,-175.690,7.970,148.296
C03454=1224.814,411.254,-81.264,-175.690,7.973,148.297
C03455=1224.810,411.501,-81.299,-175.689,7.974,148.297
C03456=1224.805,411.749,-81.333,-175.689,7.976,148.297
C03457=1224.802,411.996,-81.368,-175.688,7.980,148.298
C03458=1224.798,412.243,-81.403,-175.687,7.982,148.298
C03459=1224.794,412.491,-81.438,-175.687,7.984,148.299
C03460=1224.790,412.738,-81.471,-175.686,7.986,148.299
C03461=1224.786,412.987,-81.506,-175.686,7.988,148.300
C03462=1224.781,413.234,-81.541,-175.686,7.990,148.300
C03463=1224.778,413.481,-81.576,-175.685,7.992,148.300
C03464=1224.773,413.729,-81.611,-175.684,7.995,148.301
C03465=1224.770,413.977,-81.645,-175.684,7.997,148.301
C03466=1224.765,414.224,-81.679,-175.683,7.999,148.302
C03467=1224.761,414.472,-81.714,-175.682,8.001,148.302
C03468=1224.757,414.719,-81.749,-175.682,8.003,148.303
C03469=1224.754,414.967,-81.784,-175.681,8.005,148.303
C03470=1224.749,415.214,-81.818,-175.681,8.007,148.303
C03471=1224.745,415.462,-81.853,-175.681,8.010,148.304
C03472=1224.738,415.870,-81.910,-175.679,8.014,148.304
C03473=1224.732,416.278,-81.967,-175.679,8.017,148.305
C03474=1224.725,416.685,-82.025,-175.677,8.021,148.306
C03475=1224.721,417.092,-82.081,-175.677,8.024,148.306
C03476=1224.300,417.092,-82.115,-175.680,8.034,148.310
C03477=1224.303,416.682,-82.058,-175.681,8.031,148.310
C03478=1224.310,416.271,-82.000,-175.682,8.027,148.309
C03479=1224.317,415.861,-81.943,-175.682,8.024,148.308
C03480=1224.323,415.451,-81.885,-175.684,8.020,148.307
C03481=1224.328,415.204,-81.851,-175.684,8.018,148.307
C03482=1224.332,414.956,-81.816,-175.684,8.016,148.306
C03483=1224.336,414.709,-81.781,-175.685,8.014,148.306
C03484=1224.339,414.461,-81.747,-175.686,8.012,148.306
C03485=1224.344,414.214,-81.712,-175.686,8.009,148.305
C03486=1224.348,413.966,-81.677,-175.687,8.007,148.305
C03487=1224.352,413.719,-81.642,-175.687,8.005,148.305
C03488=1224.356,413.471,-81.607,-175.688,8.002,148.304
C03489=1224.360,413.224,-81.573,-175.689,8.000,148.304
C03490=1224.364,412.976,-81.539,-175.689,7.998,148.303
C03491=1224.368,412.728,-81.504,-175.689,7.996,148.303
C03492=1224.372,412.481,-81.468,-175.690,7.994,148.302
C03493=1224.376,412.234,-81.435,-175.691,7.992,148.302
C03494=1224.380,411.985,-81.400,-175.691,7.990,148.302
C03495=1224.384,411.738,-81.365,-175.692,7.987,148.301
C03496=1224.388,411.490,-81.330,-175.692,7.985,148.301
C03497=1224.392,411.243,-81.297,-175.693,7.983,148.300
C03498=1224.396,410.995,-81.262,-175.694,7.981,148.300
C03499=1224.400,410.748,-81.227,-175.694,7.979,148.299
C03500=1224.404,410.501,-81.193,-175.694,7.977,148.299
C03501=1224.408,410.253,-81.158,-175.696,7.974,148.299
C03502=1224.413,410.005,-81.123,-175.696,7.972,148.298
C03503=1224.417,409.757,-81.089,-175.696,7.970,148.298
C03504=1224.420,409.510,-81.055,-175.697,7.968,148.297
C03505=1224.424,409.262,-81.020,-175.697,7.965,148.297
C03506=1224.429,409.015,-80.985,-175.698,7.963,148.297
C03507=1224.432,408.767,-80.950,-175.699,7.960,148.296
C03508=1224.436,408.520,-80.916,-175.699,7.958,148.296
C03509=1224.441,408.272,-80.882,-175.700,7.956,148.295
C03510=1224.444,408.025,-80.847,-175.700,7.954,148.295
C03511=1224.449,407.777,-80.813,-175.701,7.951,148.294
C03512=1224.453,407.529,-80.778,-175.702,7.949,148.294
C03513=1224.457,407.282,-80.744,-175.702,7.947,148.293
C03514=1224.461,407.034,-80.709,-175.703,7.945,148.293
C03515=1224.465,406.786,-80.675,-175.703,7.943,148.293
C03516=1224.470,406.539,-80.640,-175.704,7.940,148.292
C03517=1224.473,406.291,-80.606,-175.705,7.938,148.292
C03518=1224.478,406.044,-80.572,-175.705,7.936,148.291
C03519=1224.482,405.796,-80.537,-175.705,7.934,148.291
C03520=1224.485,405.549,-80.503,-175.707,7.931,148.291
C03521=1224.490,405.301,-80.469,-175.707,7.929,148.290
C03522=1224.493,405.053,-80.434,-175.707,7.927,148.290
C03523=1224.498,404.806,-80.400,-175.709,7.924,148.289
C03524=1224.502,404.558,-80.365,-175.709,7.921,148.289
C03525=1224.506,404.311,-80.331,-175.709,7.919,148.288
C03526=1224.510,404.063,-80.297,-175.710,7.918,148.288
C03527=1224.514,403.815,-80.262,-175.711,7.914,148.287
C03528=1224.518,403.568,-80.228,-175.711,7.912,148.287
C03529=1224.522,403.320,-80.193,-175.712,7.910,148.287
C03530=1224.526,403.073,-80.159,-175.713,7.907,148.286
C03531=1224.530,402.825,-80.125,-175.713,7.905,148.286
C03532=1224.534,402.577,-80.090,-175.714,7.903,148.285
C03533=1224.538,402.330,-80.056,-175.715,7.900,148.285
C03534=1224.542,402.082,-80.021,-175.715,7.898,148.285
C03535=1224.546,401.835,-79.987,-175.716,7.896,148.284
C03536=1224.550,401.588,-79.953,-175.717,7.893,148.284
C03537=1224.554,401.339,-79.918,-175.717,7.891,148.283
C03538=1224.559,401.092,-79.885,-175.718,7.889,148.283
C03539=1224.563,400.844,-79.850,-175.719,7.886,148.282
C03540=1224.566,400.596,-79.816,-175.719,7.884,148.282
C03541=1224.571,400.349,-79.782,-175.720,7.882,148.281
C03542=1224.575,400.102,-79.748,-175.721,7.879,148.281
C03543=1224.579,399.854,-79.713,-175.721,7.877,148.281
C03544=1224.583,399.606,-79.679,-175.722,7.875,148.280
C03545=1224.587,399.359,-79.645,-175.723,7.872,148.280
C03546=1224.591,399.111,-79.611,-175.723,7.870,148.279
C03547=1224.595,398.863,-79.577,-175.724,7.867,148.279
C03548=1224.599,398.615,-79.542,-175.725,7.865,148.278
C03549=1224.603,398.368,-79.508,-175.725,7.863,148.278
C03550=1224.608,398.121,-79.474,-175.727,7.860,148.278
C03551=1224.611,397.873,-79.439,-175.727,7.858,148.277
C03552=1224.616,397.625,-79.406,-175.728,7.855,148.277
C03553=1224.620,397.378,-79.372,-175.729,7.853,148.276
C03554=1224.624,397.130,-79.337,-175.729,7.850,148.276
C03555=1224.627,396.883,-79.303,-175.730,7.848,148.275
C03556=1224.632,396.635,-79.268,-175.731,7.846,148.275
C03557=1224.636,396.387,-79.235,-175.731,7.843,148.275
C03558=1224.640,396.139,-79.201,-175.732,7.841,148.274
C03559=1224.644,395.892,-79.167,-175.733,7.838,148.274
C03560=1224.648,395.645,-79.132,-175.734,7.836,148.273
C03561=1224.652,395.396,-79.099,-175.735,7.833,148.273
C03562=1224.657,395.149,-79.064,-175.735,7.831,148.273
C03563=1224.660,394.902,-79.030,-175.736,7.828,148.272
C03564=1224.664,394.654,-78.995,-175.737,7.826,148.272
C03565=1224.668,394.406,-78.962,-175.738,7.823,148.271
C03566=1224.673,394.159,-78.928,-175.738,7.821,148.271
C03567=1224.676,393.911,-78.894,-175.740,7.818,148.270
C03568=1224.681,393.663,-78.860,-175.740,7.816,148.270
C03569=1224.685,393.381,-78.821,-175.741,7.813,148.269
C03570=1224.690,393.101,-78.783,-175.742,7.810,148.269
C03571=1224.695,392.819,-78.744,-175.743,7.807,148.268
C03572=1224.699,392.537,-78.705,-175.744,7.804,148.268
C03573=1224.703,392.289,-78.672,-175.744,7.802,148.268
C03574=1224.707,392.041,-78.637,-175.745,7.799,148.267
C03575=1224.711,391.794,-78.603,-175.746,7.797,148.267
C03576=1224.716,391.546,-78.569,-175.747,7.795,148.266
C03577=1224.720,391.299,-78.535,-175.747,7.792,148.266
C03578=1224.723,391.051,-78.501,-175.748,7.789,148.265
C03579=1224.728,390.803,-78.467,-175.750,7.787,148.265
C03580=1224.732,390.556,-78.434,-175.750,7.785,148.265
C03581=1224.736,390.307,-78.399,-175.751,7.782,148.264
C03582=1224.740,390.060,-78.366,-175.752,7.780,148.264
C03583=1224.744,389.813,-78.332,-175.753,7.777,148.263
C03584=1224.749,389.565,-78.298,-175.754,7.774,148.263
C03585=1224.752,389.317,-78.264,-175.755,7.772,148.263
C03586=1224.757,389.069,-78.230,-175.756,7.769,148.262
C03587=1224.761,388.822,-78.196,-175.756,7.767,148.262
C03588=1224.765,388.574,-78.163,-175.757,7.764,148.261
C03589=1224.769,388.326,-78.128,-175.758,7.761,148.261
C03590=1224.773,388.079,-78.095,-175.759,7.759,148.261
C03591=1224.777,387.831,-78.061,-175.760,7.756,148.260
C03592=1224.781,387.584,-78.027,-175.761,7.754,148.260
C03593=1224.785,387.336,-77.993,-175.761,7.751,148.259
C03594=1224.789,387.089,-77.959,-175.763,7.748,148.259
C03595=1224.794,386.840,-77.925,-175.764,7.746,148.258
C03596=1224.797,386.593,-77.892,-175.764,7.744,148.258
C03597=1224.802,386.346,-77.858,-175.766,7.741,148.258
C03598=1224.806,386.097,-77.824,-175.767,7.738,148.257
C03599=1224.810,385.850,-77.790,-175.767,7.736,148.257
C03600=1224.814,385.602,-77.757,-175.768,7.733,148.256
C03601=1224.818,385.355,-77.723,-175.769,7.730,148.256
C03602=1224.823,385.107,-77.690,-175.770,7.728,148.256
C03603=1224.826,384.859,-77.655,-175.771,7.725,148.255
C03604=1224.830,384.611,-77.622,-175.772,7.722,148.255
C03605=1224.834,384.364,-77.588,-175.773,7.720,148.254
C03606=1224.839,384.116,-77.555,-175.774,7.718,148.254
C03607=1224.843,383.869,-77.522,-175.775,7.715,148.254
C03608=1224.847,383.621,-77.488,-175.776,7.712,148.253
C03609=1224.851,383.373,-77.454,-175.778,7.709,148.253
C03610=1224.855,383.126,-77.420,-175.778,7.707,148.252
C03611=1224.859,382.878,-77.387,-175.779,7.704,148.252
C03612=1224.863,382.630,-77.353,-175.780,7.701,148.252
C03613=1224.868,382.383,-77.319,-175.781,7.698,148.251
C03614=1224.872,382.135,-77.286,-175.782,7.696,148.251
C03615=1224.875,381.887,-77.252,-175.783,7.694,148.250
C03616=1224.879,381.639,-77.218,-175.784,7.691,148.250
C03617=1224.884,381.391,-77.185,-175.785,7.688,148.250
C03618=1224.888,381.144,-77.151,-175.787,7.685,148.249
C03619=1224.892,380.897,-77.118,-175.787,7.683,148.249
C03620=1224.896,380.649,-77.084,-175.788,7.680,148.248
C03621=1224.900,380.400,-77.051,-175.790,7.678,148.248
C03622=1224.904,380.153,-77.016,-175.791,7.675,148.248
C03623=1224.908,379.905,-76.983,-175.792,7.672,148.247
C03624=1224.912,379.657,-76.950,-175.793,7.670,148.247
C03625=1224.917,379.410,-76.917,-175.794,7.667,148.247
C03626=1224.920,379.163,-76.883,-175.795,7.664,148.246
C03627=1224.925,378.915,-76.849,-175.796,7.661,148.246
C03628=1224.929,378.667,-76.816,-175.797,7.659,148.245
C03629=1224.933,378.418,-76.783,-175.798,7.656,148.245
C03630=1224.937,378.171,-76.749,-175.799,7.654,148.245
C03631=1224.941,377.924,-76.716,-175.801,7.651,148.244
C03632=1224.945,377.676,-76.682,-175.802,7.649,148.244
C03633=1224.949,377.428,-76.649,-175.803,7.646,148.244
C03634=1224.954,377.180,-76.616,-175.804,7.643,148.243
C03635=1224.958,376.932,-76.582,-175.805,7.640,148.243
C03636=1224.962,376.685,-76.549,-175.807,7.637,148.242
C03637=1224.966,376.438,-76.515,-175.808,7.634,148.242
C03638=1224.970,376.190,-76.482,-175.808,7.632,148.242
C03639=1224.974,375.941,-76.449,-175.810,7.630,148.241
C03640=1224.978,375.694,-76.416,-175.811,7.627,148.241
C03641=1224.982,375.446,-76.382,-175.812,7.624,148.241
C03642=1224.986,375.198,-76.349,-175.814,7.621,148.240
C03643=1224.990,374.951,-76.315,-175.815,7.619,148.240
C03644=1224.994,374.703,-76.282,-175.816,7.616,148.239
C03645=1224.999,374.455,-76.248,-175.817,7.613,148.239
C03646=1225.003,374.208,-76.215,-175.819,7.610,148.239
C03647=1225.007,373.960,-76.182,-175.820,7.608,148.239
C03648=1225.011,373.712,-76.149,-175.821,7.605,148.238
C03649=1225.016,373.464,-76.116,-175.822,7.602,148.238
C03650=1225.020,373.217,-76.083,-175.823,7.599,148.237
